Universal Robots PolyScope program: faichun_9jan_1t1.urp

Program faichun_9jan_1t1 (installation=default directory=/programs createdIn=5.11.9.1010452 lastSavedIn=5.11.9.1010452 robotSerialNumber=20225200364)
Calibrated DH parameters: a=[0.00002, -0.569483, -0.54992, -0.00001, -0.000036, 0]; d=[0.180894, -146.691669, 192.918669, -46.053088, 0.119778, 0.115602]; alpha=[1.571425, -0.001534, 0.003359, 1.568739, -1.571477, 0]; deltaTheta=[0, 0.376258, -0.101074, -0.275185, -0.000002, 0]
Robot Program (runOnlyOnce=true)
  Script file /programs/FaiChun_9 Jan_11_2_t1.script
    | def Machining1():
    |   # Default parameters:
    |   global speed_ms = 0.05
    |   global speed_rads = 0.75
    |   global accel_mss = 3
    |   global accel_radss = 1.2
    |   global blend_radius_m = 0.0003
    | 
    |   # Add subprograms here
    |   # Start of main program
    |   # Program generated by RoboDK v5.6.8 for UR10e on 17/01/2025 15:24:14
    |   # Using nominal kinematics.
    |   blend_radius_m = 0.0003
    |   speed_ms = 0.05
    |   # set_reference(p[0.340000, -0.240000, 0.001500, 0.000000, 0.000000, 0.000000])
    |   set_tcp(p[0.000000, 0.000000, 0.252000, 0.000000, 0.000000, 0.000000])
    |   # Show Tool
    |   movej([0.140721, -1.398447, -2.445688, -0.868253, 1.570796, 1.711517],accel_radss,speed_rads,0,blend_radius_m)
    |   movel([0.140721, -1.451124, -2.475554, -0.785711, 1.570796, 1.711517],accel_mss,speed_ms,0,blend_radius_m)
    |   #SetTool1
    |   #M_RunCode6
    |   #SetRPM60000
    |   speed_ms = 0.05
    |   #M_RunCode3
    |   movel([0.140721, -1.474076, -2.486639, -0.751674, 1.570796, 1.711517],accel_mss,speed_ms,0,blend_radius_m)
    |   speed_ms = 0.003
    |   movel([0.140721, -1.480003, -2.489338, -0.743048, 1.570796, 1.711517],accel_mss,speed_ms,0,blend_radius_m)
    |   speed_ms = 0.02
    |   movel([-0.135603, -1.563113, -2.412732, -0.736544, 1.570796, 1.435194],accel_mss,speed_ms,0,blend_radius_m)
    |   movel([-0.182919, -1.334068, -2.598334, -0.779987, 1.570796, 1.387878],accel_mss,speed_ms,0,blend_radius_m)
    |   movel([0.198662, -1.168946, -2.687374, -0.856069, 1.570796, 1.769459],accel_mss,speed_ms,0,blend_radius_m)
    |   movel([0.140721, -1.480003, -2.489338, -0.743048, 1.570796, 1.711517],accel_mss,speed_ms,0,blend_radius_m)
    |   speed_ms = 0.003
    |   movel([0.140721, -1.474076, -2.486639, -0.751674, 1.570796, 1.711517],accel_mss,speed_ms,0,blend_radius_m)
    |   speed_ms = 0.05
    |   movel([0.140721, -1.451124, -2.475554, -0.785711, 1.570796, 1.711517],accel_mss,speed_ms,0,blend_radius_m)
    |   #M_RunCode9
    |   movel([0.136570, -1.444454, -2.480985, -0.786951, 1.570796, 1.707367],accel_mss,speed_ms,0,blend_radius_m)
    |   #M_RunCode3
    |   movel([0.136570, -1.467543, -2.492148, -0.752698, 1.570796, 1.707367],accel_mss,speed_ms,0,blend_radius_m)
    |   speed_ms = 0.003
    |   movel([0.136570, -1.473508, -2.494867, -0.744014, 1.570796, 1.707367],accel_mss,speed_ms,0,blend_radius_m)
    |   speed_ms = 0.012
    |   movel([0.132210, -1.474416, -2.494098, -0.743875, 1.570796, 1.703007],accel_mss,speed_ms,0,blend_radius_m)
    |   movel([0.131633, -1.478168, -2.490906, -0.743314, 1.570796, 1.702429],accel_mss,speed_ms,0,blend_radius_m)
    |   movel([0.125209, -1.479526, -2.489746, -0.743117, 1.570796, 1.696006],accel_mss,speed_ms,0,blend_radius_m)
    |   movel([0.125756, -1.475786, -2.492935, -0.743668, 1.570796, 1.696552],accel_mss,speed_ms,0,blend_radius_m)
    |   movel([0.123495, -1.476273, -2.492521, -0.743595, 1.570796, 1.694292],accel_mss,speed_ms,0,blend_radius_m)
    |   movel([0.122957, -1.480010, -2.489332, -0.743047, 1.570796, 1.693753],accel_mss,speed_ms,0,blend_radius_m)
    |   movel([0.117581, -1.481181, -2.488328, -0.742880, 1.570796, 1.688377],accel_mss,speed_ms,0,blend_radius_m)
    |   movel([0.116539, -1.481408, -2.488133, -0.742848, 1.570796, 1.687335],accel_mss,speed_ms,0,blend_radius_m)
    |   movel([0.117294, -1.475890, -2.492847, -0.743652, 1.570796, 1.688091],accel_mss,speed_ms,0,blend_radius_m)
    |   movel([0.121657, -1.474929, -2.493663, -0.743797, 1.570796, 1.692454],accel_mss,speed_ms,0,blend_radius_m)
    |   movel([0.121935, -1.472979, -2.495315, -0.744096, 1.570796, 1.692731],accel_mss,speed_ms,0,blend_radius_m)
    |   movel([0.115294, -1.474450, -2.494069, -0.743870, 1.570796, 1.686091],accel_mss,speed_ms,0,blend_radius_m)
    |   movel([0.114291, -1.481907, -2.487705, -0.742777, 1.570796, 1.685087],accel_mss,speed_ms,0,blend_radius_m)
    |   movel([0.113249, -1.482141, -2.487504, -0.742744, 1.570796, 1.684045],accel_mss,speed_ms,0,blend_radius_m)
    |   speed_ms = 0.02
    |   movel([-0.001403, -1.512452, -2.460728, -0.739209, 1.570796, 1.569393],accel_mss,speed_ms,0,blend_radius_m)
    |   movel([-0.112335, -1.550651, -2.424918, -0.736820, 1.570796, 1.458461],accel_mss,speed_ms,0,blend_radius_m)
    |   speed_ms = 0.012
    |   movel([-0.113250, -1.544354, -2.430981, -0.737054, 1.570796, 1.457547],accel_mss,speed_ms,0,blend_radius_m)
    |   movel([-0.119333, -1.546716, -2.428713, -0.736959, 1.570796, 1.451463],accel_mss,speed_ms,0,blend_radius_m)
    |   movel([-0.119087, -1.548345, -2.427145, -0.736899, 1.570796, 1.451710],accel_mss,speed_ms,0,blend_radius_m)
    |   movel([-0.115090, -1.546793, -2.428639, -0.736956, 1.570796, 1.455706],accel_mss,speed_ms,0,blend_radius_m)
    |   movel([-0.114409, -1.551442, -2.424151, -0.736796, 1.570796, 1.456387],accel_mss,speed_ms,0,blend_radius_m)
    |   movel([-0.115366, -1.551811, -2.423794, -0.736784, 1.570796, 1.455430],accel_mss,speed_ms,0,blend_radius_m)
    |   movel([-0.120291, -1.553718, -2.421942, -0.736729, 1.570796, 1.450506],accel_mss,speed_ms,0,blend_radius_m)
    |   movel([-0.120772, -1.550599, -2.424968, -0.736822, 1.570796, 1.450025],accel_mss,speed_ms,0,blend_radius_m)
    |   movel([-0.122835, -1.551404, -2.424188, -0.736797, 1.570796, 1.447961],accel_mss,speed_ms,0,blend_radius_m)
    |   movel([-0.122346, -1.554519, -2.421162, -0.736708, 1.570796, 1.448450],accel_mss,speed_ms,0,blend_radius_m)
    |   movel([-0.128198, -1.556814, -2.418922, -0.736653, 1.570796, 1.442598],accel_mss,speed_ms,0,blend_radius_m)
    |   movel([-0.128709, -1.553718, -2.421941, -0.736729, 1.570796, 1.442088],accel_mss,speed_ms,0,blend_radius_m)
    |   movel([-0.132665, -1.555290, -2.420410, -0.736688, 1.570796, 1.438132],accel_mss,speed_ms,0,blend_radius_m)
    |   movel([-0.133450, -1.550705, -2.424865, -0.736819, 1.570796, 1.437347],accel_mss,speed_ms,0,blend_radius_m)
    |   movel([-0.129474, -1.549116, -2.426401, -0.736872, 1.570796, 1.441323],accel_mss,speed_ms,0,blend_radius_m)
    |   movel([-0.129743, -1.547498, -2.427961, -0.736930, 1.570796, 1.441053],accel_mss,speed_ms,0,blend_radius_m)
    |   movel([-0.133727, -1.549091, -2.426425, -0.736873, 1.570796, 1.437069],accel_mss,speed_ms,0,blend_radius_m)
    |   movel([-0.134396, -1.545231, -2.430140, -0.737018, 1.570796, 1.436400],accel_mss,speed_ms,0,blend_radius_m)
    |   movel([-0.134524, -1.544477, -2.430863, -0.737049, 1.570796, 1.436272],accel_mss,speed_ms,0,blend_radius_m)
    |   movel([-0.128589, -1.542092, -2.433143, -0.737154, 1.570796, 1.442208],accel_mss,speed_ms,0,blend_radius_m)
    |   movel([-0.128072, -1.545228, -2.430143, -0.737018, 1.570796, 1.442725],accel_mss,speed_ms,0,blend_radius_m)
    |   movel([-0.125992, -1.544401, -2.430936, -0.737052, 1.570796, 1.444805],accel_mss,speed_ms,0,blend_radius_m)
    |   movel([-0.126769, -1.539625, -2.435492, -0.737272, 1.570796, 1.444027],accel_mss,speed_ms,0,blend_radius_m)
    |   movel([-0.134806, -1.542853, -2.432416, -0.737120, 1.570796, 1.435990],accel_mss,speed_ms,0,blend_radius_m)
    |   movel([-0.151268, -1.454119, -2.510984, -0.747286, 1.570796, 1.419528],accel_mss,speed_ms,0,blend_radius_m)
    |   speed_ms = 0.02
    |   movel([-0.171874, -1.356528, -2.583560, -0.772301, 1.570796, 1.398922],accel_mss,speed_ms,0,blend_radius_m)
    |   movel([-0.172081, -1.355600, -2.584184, -0.772605, 1.570796, 1.398715],accel_mss,speed_ms,0,blend_radius_m)
    |   speed_ms = 0.012
    |   movel([-0.162028, -1.350393, -2.587664, -0.774332, 1.570796, 1.408769],accel_mss,speed_ms,0,blend_radius_m)
    |   movel([-0.163290, -1.344436, -2.591600, -0.776353, 1.570796, 1.407507],accel_mss,speed_ms,0,blend_radius_m)
    |   movel([-0.165922, -1.345805, -2.590700, -0.775884, 1.570796, 1.404874],accel_mss,speed_ms,0,blend_radius_m)
    |   movel([-0.165080, -1.349718, -2.588113, -0.774558, 1.570796, 1.405716],accel_mss,speed_ms,0,blend_radius_m)
    |   movel([-0.172527, -1.353588, -2.585533, -0.773268, 1.570796, 1.398269],accel_mss,speed_ms,0,blend_radius_m)
    |   movel([-0.172737, -1.352660, -2.586154, -0.773575, 1.570796, 1.398059],accel_mss,speed_ms,0,blend_radius_m)
    |   movel([-0.173831, -1.347848, -2.589351, -0.775189, 1.570796, 1.396966],accel_mss,speed_ms,0,blend_radius_m)
    |   movel([-0.168773, -1.345194, -2.591101, -0.776093, 1.570796, 1.402023],accel_mss,speed_ms,0,blend_radius_m)
    |   movel([-0.169223, -1.343160, -2.592436, -0.776792, 1.570796, 1.401574],accel_mss,speed_ms,0,blend_radius_m)
    |   movel([-0.174292, -1.345828, -2.590684, -0.775876, 1.570796, 1.396505],accel_mss,speed_ms,0,blend_radius_m)
    |   movel([-0.175621, -1.340037, -2.594475, -0.777877, 1.570796, 1.395175],accel_mss,speed_ms,0,blend_radius_m)
    |   movel([-0.170518, -1.337328, -2.596232, -0.778829, 1.570796, 1.400279],accel_mss,speed_ms,0,blend_radius_m)
    |   movel([-0.171402, -1.333368, -2.598783, -0.780238, 1.570796, 1.399394],accel_mss,speed_ms,0,blend_radius_m)
    |   movel([-0.163769, -1.329319, -2.601369, -0.781700, 1.570796, 1.407028],accel_mss,speed_ms,0,blend_radius_m)
    |   movel([-0.162919, -1.333321, -2.598813, -0.780255, 1.570796, 1.407878],accel_mss,speed_ms,0,blend_radius_m)
    |   movel([-0.160246, -1.331919, -2.599711, -0.780759, 1.570796, 1.410551],accel_mss,speed_ms,0,blend_radius_m)
    |   movel([-0.161083, -1.327903, -2.602269, -0.782217, 1.570796, 1.409713],accel_mss,speed_ms,0,blend_radius_m)
    |   movel([-0.153386, -1.323865, -2.604819, -0.783706, 1.570796, 1.417410],accel_mss,speed_ms,0,blend_radius_m)
    |   movel([-0.152202, -1.329868, -2.601020, -0.781501, 1.570796, 1.418594],accel_mss,speed_ms,0,blend_radius_m)
    |   movel([-0.157369, -1.332552, -2.599306, -0.780531, 1.570796, 1.413427],accel_mss,speed_ms,0,blend_radius_m)
    |   movel([-0.156945, -1.334634, -2.597970, -0.779785, 1.570796, 1.413851],accel_mss,speed_ms,0,blend_radius_m)
    |   movel([-0.149106, -1.330580, -2.600566, -0.781243, 1.570796, 1.421690],accel_mss,speed_ms,0,blend_radius_m)
    |   movel([-0.150679, -1.322452, -2.605705, -0.784232, 1.570796, 1.420118],accel_mss,speed_ms,0,blend_radius_m)
    |   movel([-0.001924, -1.251119, -2.647144, -0.814126, 1.570796, 1.568873],accel_mss,speed_ms,0,blend_radius_m)
    |   speed_ms = 0.02
    |   movel([0.158957, -1.188696, -2.678386, -0.845308, 1.570796, 1.729754],accel_mss,speed_ms,0,blend_radius_m)
    |   movel([0.157034, -1.200160, -2.672976, -0.839253, 1.570796, 1.727831],accel_mss,speed_ms,0,blend_radius_m)
    |   speed_ms = 0.012
    |   movel([0.166189, -1.197160, -2.674405, -0.840823, 1.570796, 1.736986],accel_mss,speed_ms,0,blend_radius_m)
    |   movel([0.166716, -1.194184, -2.675814, -0.842391, 1.570796, 1.737513],accel_mss,speed_ms,0,blend_radius_m)
    |   movel([0.160669, -1.196167, -2.674876, -0.841345, 1.570796, 1.731466],accel_mss,speed_ms,0,blend_radius_m)
    |   movel([0.162134, -1.187639, -2.678877, -0.845873, 1.570796, 1.732930],accel_mss,speed_ms,0,blend_radius_m)
    |   movel([0.163603, -1.187149, -2.679104, -0.846136, 1.570796, 1.734399],accel_mss,speed_ms,0,blend_radius_m)
    |   movel([0.171178, -1.184645, -2.680263, -0.847481, 1.570796, 1.741974],accel_mss,speed_ms,0,blend_radius_m)
    |   movel([0.170131, -1.190457, -2.677564, -0.844368, 1.570796, 1.740927],accel_mss,speed_ms,0,blend_radius_m)
    |   movel([0.173284, -1.189438, -2.678039, -0.844911, 1.570796, 1.744080],accel_mss,speed_ms,0,blend_radius_m)
    |   movel([0.174358, -1.183606, -2.680741, -0.848041, 1.570796, 1.745154],accel_mss,speed_ms,0,blend_radius_m)
    |   movel([0.183424, -1.180682, -2.682083, -0.849624, 1.570796, 1.754220],accel_mss,speed_ms,0,blend_radius_m)
    |   movel([0.182294, -1.186557, -2.679379, -0.846453, 1.570796, 1.753091],accel_mss,speed_ms,0,blend_radius_m)
    |   movel([0.188385, -1.184641, -2.680265, -0.847483, 1.570796, 1.759181],accel_mss,speed_ms,0,blend_radius_m)
    |   movel([0.186680, -1.193280, -2.676240, -0.842870, 1.570796, 1.757477],accel_mss,speed_ms,0,blend_radius_m)
    |   movel([0.180648, -1.195154, -2.675356, -0.841879, 1.570796, 1.751444],accel_mss,speed_ms,0,blend_radius_m)
    |   movel([0.180078, -1.198139, -2.673940, -0.840310, 1.570796, 1.750875],accel_mss,speed_ms,0,blend_radius_m)
    |   movel([0.186090, -1.196283, -2.674822, -0.841285, 1.570796, 1.756886],accel_mss,speed_ms,0,blend_radius_m)
    |   movel([0.184696, -1.203394, -2.671424, -0.837571, 1.570796, 1.755493],accel_mss,speed_ms,0,blend_radius_m)
    |   movel([0.184428, -1.204765, -2.670763, -0.836861, 1.570796, 1.755225],accel_mss,speed_ms,0,blend_radius_m)
    |   movel([0.175610, -1.207468, -2.669453, -0.835468, 1.570796, 1.746407],accel_mss,speed_ms,0,blend_radius_m)
    |   movel([0.176673, -1.201793, -2.672194, -0.838402, 1.570796, 1.747469],accel_mss,speed_ms,0,blend_radius_m)
    |   movel([0.173563, -1.202767, -2.671726, -0.837896, 1.570796, 1.744359],accel_mss,speed_ms,0,blend_radius_m)
    |   movel([0.171983, -1.211350, -2.667557, -0.833482, 1.570796, 1.742780],accel_mss,speed_ms,0,blend_radius_m)
    |   movel([0.183853, -1.207714, -2.669333, -0.835342, 1.570796, 1.754649],accel_mss,speed_ms,0,blend_radius_m)
    |   speed_ms = 0.02
    |   movel([0.158243, -1.345021, -2.591215, -0.776152, 1.570796, 1.729039],accel_mss,speed_ms,0,blend_radius_m)
    |   movel([0.139022, -1.458254, -2.507595, -0.746540, 1.570796, 1.709818],accel_mss,speed_ms,0,blend_radius_m)
    |   speed_ms = 0.012
    |   movel([0.130132, -1.460164, -2.506021, -0.746204, 1.570796, 1.700928],accel_mss,speed_ms,0,blend_radius_m)
    |   movel([0.129256, -1.465966, -2.501205, -0.745218, 1.570796, 1.700052],accel_mss,speed_ms,0,blend_radius_m)
    |   movel([0.131545, -1.465473, -2.501616, -0.745300, 1.570796, 1.702341],accel_mss,speed_ms,0,blend_radius_m)
    |   movel([0.132131, -1.461656, -2.504788, -0.745945, 1.570796, 1.702927],accel_mss,speed_ms,0,blend_radius_m)
    |   movel([0.138690, -1.460258, -2.505944, -0.746187, 1.570796, 1.709487],accel_mss,speed_ms,0,blend_radius_m)
    |   movel([0.138542, -1.461182, -2.505180, -0.746027, 1.570796, 1.709338],accel_mss,speed_ms,0,blend_radius_m)
    |   movel([0.137780, -1.465926, -2.501239, -0.745225, 1.570796, 1.708576],accel_mss,speed_ms,0,blend_radius_m)
    |   movel([0.133380, -1.466851, -2.500465, -0.745072, 1.570796, 1.704177],accel_mss,speed_ms,0,blend_radius_m)
    |   movel([0.133075, -1.468822, -2.498815, -0.744752, 1.570796, 1.703871],accel_mss,speed_ms,0,blend_radius_m)
    |   movel([0.137466, -1.467900, -2.499588, -0.744901, 1.570796, 1.708263],accel_mss,speed_ms,0,blend_radius_m)
    |   movel([0.136570, -1.473508, -2.494867, -0.744014, 1.570796, 1.707367],accel_mss,speed_ms,0,blend_radius_m)
    |   speed_ms = 0.003
    |   movel([0.136570, -1.467543, -2.492148, -0.752698, 1.570796, 1.707367],accel_mss,speed_ms,0,blend_radius_m)
    |   speed_ms = 0.05
    |   movel([0.136570, -1.444454, -2.480985, -0.786951, 1.570796, 1.707367],accel_mss,speed_ms,0,blend_radius_m)
    |   #M_RunCode9
    |   movel([-0.101116, -1.322556, -2.569102, -0.820731, 1.570796, 1.469680],accel_mss,speed_ms,0,blend_radius_m)
    |   #M_RunCode3
    |   # num 0 inside
    |   movel([-0.101116, -1.347956, -2.581781, -0.782652, 1.570796, 1.469680],accel_mss,speed_ms,0,blend_radius_m)
    |   speed_ms = 0.003
    |   movel([-0.101116, -1.354564, -2.584879, -0.772945, 1.570796, 1.469680],accel_mss,speed_ms,0,blend_radius_m)
    |   speed_ms = 0.015
    |   movel([-0.106161, -1.361335, -2.580307, -0.770747, 1.570796, 1.464635],accel_mss,speed_ms,0,blend_radius_m)
    |   movel([-0.110090, -1.365943, -2.577159, -0.769287, 1.570796, 1.460707],accel_mss,speed_ms,0,blend_radius_m)
    |   movel([-0.111700, -1.367455, -2.576119, -0.768814, 1.570796, 1.459096],accel_mss,speed_ms,0,blend_radius_m)
    |   movel([-0.113150, -1.368443, -2.575438, -0.768507, 1.570796, 1.457647],accel_mss,speed_ms,0,blend_radius_m)
    |   movel([-0.114438, -1.368913, -2.575114, -0.768362, 1.570796, 1.456358],accel_mss,speed_ms,0,blend_radius_m)
    |   movel([-0.115571, -1.368864, -2.575148, -0.768377, 1.570796, 1.455226],accel_mss,speed_ms,0,blend_radius_m)
    |   movel([-0.116374, -1.368348, -2.575504, -0.768537, 1.570796, 1.454422],accel_mss,speed_ms,0,blend_radius_m)
    |   movel([-0.116674, -1.367414, -2.576148, -0.768827, 1.570796, 1.454122],accel_mss,speed_ms,0,blend_radius_m)
    |   movel([-0.116470, -1.366059, -2.577080, -0.769251, 1.570796, 1.454326],accel_mss,speed_ms,0,blend_radius_m)
    |   movel([-0.115761, -1.364279, -2.578299, -0.769810, 1.570796, 1.455035],accel_mss,speed_ms,0,blend_radius_m)
    |   movel([-0.112933, -1.359327, -2.581670, -0.771392, 1.570796, 1.457863],accel_mss,speed_ms,0,blend_radius_m)
    |   movel([-0.108281, -1.352413, -2.586319, -0.773657, 1.570796, 1.462515],accel_mss,speed_ms,0,blend_radius_m)
    |   movel([-0.103194, -1.345531, -2.590880, -0.775978, 1.570796, 1.467603],accel_mss,speed_ms,0,blend_radius_m)
    |   movel([-0.099141, -1.340763, -2.594002, -0.777624, 1.570796, 1.471655],accel_mss,speed_ms,0,blend_radius_m)
    |   movel([-0.097464, -1.339187, -2.595027, -0.778175, 1.570796, 1.473333],accel_mss,speed_ms,0,blend_radius_m)
    |   movel([-0.095957, -1.338153, -2.595698, -0.778538, 1.570796, 1.474840],accel_mss,speed_ms,0,blend_radius_m)
    |   movel([-0.094620, -1.337665, -2.596014, -0.778710, 1.570796, 1.476176],accel_mss,speed_ms,0,blend_radius_m)
    |   movel([-0.093457, -1.337724, -2.595976, -0.778689, 1.570796, 1.477339],accel_mss,speed_ms,0,blend_radius_m)
    |   movel([-0.092647, -1.338276, -2.595618, -0.778495, 1.570796, 1.478149],accel_mss,speed_ms,0,blend_radius_m)
    |   movel([-0.092365, -1.339263, -2.594978, -0.778148, 1.570796, 1.478432],accel_mss,speed_ms,0,blend_radius_m)
    |   movel([-0.092614, -1.340685, -2.594053, -0.777651, 1.570796, 1.478183],accel_mss,speed_ms,0,blend_radius_m)
    |   movel([-0.093386, -1.342532, -2.592847, -0.777009, 1.570796, 1.477410],accel_mss,speed_ms,0,blend_radius_m)
    |   movel([-0.096363, -1.347612, -2.589507, -0.775269, 1.570796, 1.474433],accel_mss,speed_ms,0,blend_radius_m)
    |   movel([-0.101116, -1.354564, -2.584879, -0.772945, 1.570796, 1.469680],accel_mss,speed_ms,0,blend_radius_m)
    |   speed_ms = 0.003
    |   movel([-0.101116, -1.347956, -2.581781, -0.782652, 1.570796, 1.469680],accel_mss,speed_ms,0,blend_radius_m)
    |   speed_ms = 0.05
    |   movel([-0.101116, -1.322556, -2.569102, -0.820731, 1.570796, 1.469680],accel_mss,speed_ms,0,blend_radius_m)
    |   #M_RunCode9
    |   movel([-0.093439, -1.325002, -2.567533, -0.819854, 1.570796, 1.477357],accel_mss,speed_ms,0,blend_radius_m)
    |   #M_RunCode3
    |   #num 0 outside
    |   movel([-0.093439, -1.350361, -2.580180, -0.781848, 1.570796, 1.477357],accel_mss,speed_ms,0,blend_radius_m)
    |   speed_ms = 0.003
    |   movel([-0.093439, -1.356958, -2.583270, -0.772161, 1.570796, 1.477357],accel_mss,speed_ms,0,blend_radius_m)
    |   speed_ms = 0.015
    |   movel([-0.095323, -1.359406, -2.581617, -0.771367, 1.570796, 1.475474],accel_mss,speed_ms,0,blend_radius_m)
    |   movel([-0.097250, -1.361605, -2.580124, -0.770660, 1.570796, 1.473546],accel_mss,speed_ms,0,blend_radius_m)
    |   movel([-0.099225, -1.363562, -2.578790, -0.770037, 1.570796, 1.471571],accel_mss,speed_ms,0,blend_radius_m)
    |   movel([-0.101247, -1.365276, -2.577617, -0.769496, 1.570796, 1.469549],accel_mss,speed_ms,0,blend_radius_m)
    |   movel([-0.103277, -1.366737, -2.576613, -0.769038, 1.570796, 1.467519],accel_mss,speed_ms,0,blend_radius_m)
    |   movel([-0.105274, -1.367936, -2.575788, -0.768665, 1.570796, 1.465522],accel_mss,speed_ms,0,blend_radius_m)
    |   movel([-0.107241, -1.368876, -2.575140, -0.768373, 1.570796, 1.463555],accel_mss,speed_ms,0,blend_radius_m)
    |   movel([-0.109177, -1.369553, -2.574672, -0.768164, 1.570796, 1.461619],accel_mss,speed_ms,0,blend_radius_m)
    |   movel([-0.111057, -1.369973, -2.574381, -0.768035, 1.570796, 1.459739],accel_mss,speed_ms,0,blend_radius_m)
    |   movel([-0.112847, -1.370143, -2.574264, -0.767982, 1.570796, 1.457949],accel_mss,speed_ms,0,blend_radius_m)
    |   movel([-0.114554, -1.370059, -2.574322, -0.768008, 1.570796, 1.456243],accel_mss,speed_ms,0,blend_radius_m)
    |   movel([-0.116176, -1.369726, -2.574552, -0.768111, 1.570796, 1.454621],accel_mss,speed_ms,0,blend_radius_m)
    |   movel([-0.117639, -1.369161, -2.574943, -0.768285, 1.570796, 1.453158],accel_mss,speed_ms,0,blend_radius_m)
    |   movel([-0.118861, -1.368389, -2.575476, -0.768524, 1.570796, 1.451935],accel_mss,speed_ms,0,blend_radius_m)
    |   movel([-0.119847, -1.367410, -2.576151, -0.768828, 1.570796, 1.450949],accel_mss,speed_ms,0,blend_radius_m)
    |   movel([-0.120593, -1.366216, -2.576972, -0.769201, 1.570796, 1.450203],accel_mss,speed_ms,0,blend_radius_m)
    |   movel([-0.121076, -1.364824, -2.577927, -0.769639, 1.570796, 1.449720],accel_mss,speed_ms,0,blend_radius_m)
    |   movel([-0.121271, -1.363244, -2.579007, -0.770138, 1.570796, 1.449525],accel_mss,speed_ms,0,blend_radius_m)
    |   movel([-0.121177, -1.361471, -2.580215, -0.770703, 1.570796, 1.449619],accel_mss,speed_ms,0,blend_radius_m)
    |   movel([-0.120789, -1.359505, -2.581549, -0.771335, 1.570796, 1.450007],accel_mss,speed_ms,0,blend_radius_m)
    |   movel([-0.120098, -1.357373, -2.582991, -0.772026, 1.570796, 1.450698],accel_mss,speed_ms,0,blend_radius_m)
    |   movel([-0.119085, -1.355103, -2.584518, -0.772768, 1.570796, 1.451711],accel_mss,speed_ms,0,blend_radius_m)
    |   movel([-0.117751, -1.352697, -2.586129, -0.773563, 1.570796, 1.453045],accel_mss,speed_ms,0,blend_radius_m)
    |   movel([-0.116093, -1.350152, -2.587824, -0.774413, 1.570796, 1.454704],accel_mss,speed_ms,0,blend_radius_m)
    |   movel([-0.114233, -1.347648, -2.589484, -0.775257, 1.570796, 1.456564],accel_mss,speed_ms,0,blend_radius_m)
    |   movel([-0.112304, -1.345376, -2.590982, -0.776031, 1.570796, 1.458493],accel_mss,speed_ms,0,blend_radius_m)
    |   movel([-0.110305, -1.343337, -2.592320, -0.776731, 1.570796, 1.460492],accel_mss,speed_ms,0,blend_radius_m)
    |   movel([-0.108239, -1.341537, -2.593498, -0.777355, 1.570796, 1.462557],accel_mss,speed_ms,0,blend_radius_m)
    |   movel([-0.106152, -1.339991, -2.594504, -0.777893, 1.570796, 1.464644],accel_mss,speed_ms,0,blend_radius_m)
    |   movel([-0.104092, -1.338723, -2.595328, -0.778337, 1.570796, 1.466704],accel_mss,speed_ms,0,blend_radius_m)
    |   movel([-0.102059, -1.337730, -2.595972, -0.778687, 1.570796, 1.468737],accel_mss,speed_ms,0,blend_radius_m)
    |   movel([-0.100055, -1.337017, -2.596433, -0.778939, 1.570796, 1.470741],accel_mss,speed_ms,0,blend_radius_m)
    |   movel([-0.098115, -1.336579, -2.596716, -0.779094, 1.570796, 1.472681],accel_mss,speed_ms,0,blend_radius_m)
    |   movel([-0.096266, -1.336409, -2.596826, -0.779154, 1.570796, 1.474530],accel_mss,speed_ms,0,blend_radius_m)
    |   movel([-0.094508, -1.336506, -2.596763, -0.779120, 1.570796, 1.476288],accel_mss,speed_ms,0,blend_radius_m)
    |   movel([-0.092848, -1.336874, -2.596526, -0.778989, 1.570796, 1.477948],accel_mss,speed_ms,0,blend_radius_m)
    |   movel([-0.091363, -1.337486, -2.596130, -0.778773, 1.570796, 1.479434],accel_mss,speed_ms,0,blend_radius_m)
    |   movel([-0.090132, -1.338313, -2.595594, -0.778482, 1.570796, 1.480664],accel_mss,speed_ms,0,blend_radius_m)
    |   movel([-0.089156, -1.339357, -2.594917, -0.778115, 1.570796, 1.481641],accel_mss,speed_ms,0,blend_radius_m)
    |   movel([-0.088434, -1.340616, -2.594098, -0.777675, 1.570796, 1.482363],accel_mss,speed_ms,0,blend_radius_m)
    |   movel([-0.087990, -1.342075, -2.593146, -0.777168, 1.570796, 1.482806],accel_mss,speed_ms,0,blend_radius_m)
    |   movel([-0.087851, -1.343724, -2.592067, -0.776598, 1.570796, 1.482946],accel_mss,speed_ms,0,blend_radius_m)
    |   movel([-0.088015, -1.345563, -2.590859, -0.775967, 1.570796, 1.482781],accel_mss,speed_ms,0,blend_radius_m)
    |   movel([-0.088479, -1.347585, -2.589526, -0.775279, 1.570796, 1.482317],accel_mss,speed_ms,0,blend_radius_m)
    |   movel([-0.089250, -1.349756, -2.588088, -0.774546, 1.570796, 1.481546],accel_mss,speed_ms,0,blend_radius_m)
    |   movel([-0.090337, -1.352044, -2.586565, -0.773780, 1.570796, 1.480459],accel_mss,speed_ms,0,blend_radius_m)
    |   movel([-0.091734, -1.354445, -2.584959, -0.772985, 1.570796, 1.479062],accel_mss,speed_ms,0,blend_radius_m)
    |   movel([-0.093439, -1.356958, -2.583270, -0.772161, 1.570796, 1.477357],accel_mss,speed_ms,0,blend_radius_m)
    |   speed_ms = 0.003
    |   movel([-0.093439, -1.350361, -2.580180, -0.781848, 1.570796, 1.477357],accel_mss,speed_ms,0,blend_radius_m)
    |   speed_ms = 0.05
    |   movel([-0.093439, -1.325002, -2.567533, -0.819854, 1.570796, 1.477357],accel_mss,speed_ms,0,blend_radius_m)
    |   #M_RunCode9
    |   movel([-0.123954, -1.324456, -2.567884, -0.820049, 1.570796, 1.446843],accel_mss,speed_ms,0,blend_radius_m)
    |   #M_RunCode3
    |   # num 2
    |   movel([-0.123954, -1.349824, -2.580538, -0.782027, 1.570796, 1.446843],accel_mss,speed_ms,0,blend_radius_m)
    |   speed_ms = 0.003
    |   movel([-0.123954, -1.356423, -2.583630, -0.772335, 1.570796, 1.446843],accel_mss,speed_ms,0,blend_radius_m)
    |   speed_ms = 0.02
    |   movel([-0.129998, -1.365194, -2.577673, -0.769522, 1.570796, 1.440798],accel_mss,speed_ms,0,blend_radius_m)
    |   movel([-0.153716, -1.359168, -2.581778, -0.771443, 1.570796, 1.417080],accel_mss,speed_ms,0,blend_radius_m)
    |   movel([-0.153133, -1.358284, -2.582375, -0.771729, 1.570796, 1.417664],accel_mss,speed_ms,0,blend_radius_m)
    |   movel([-0.151367, -1.356095, -2.583852, -0.772443, 1.570796, 1.419429],accel_mss,speed_ms,0,blend_radius_m)
    |   movel([-0.149072, -1.354075, -2.585207, -0.773107, 1.570796, 1.421725],accel_mss,speed_ms,0,blend_radius_m)
    |   movel([-0.146447, -1.352249, -2.586428, -0.773712, 1.570796, 1.424349],accel_mss,speed_ms,0,blend_radius_m)
    |   movel([-0.143702, -1.350644, -2.587497, -0.774248, 1.570796, 1.427094],accel_mss,speed_ms,0,blend_radius_m)
    |   movel([-0.136140, -1.346869, -2.589998, -0.775522, 1.570796, 1.434656],accel_mss,speed_ms,0,blend_radius_m)
    |   movel([-0.129079, -1.343432, -2.592258, -0.776699, 1.570796, 1.441717],accel_mss,speed_ms,0,blend_radius_m)
    |   movel([-0.126471, -1.341951, -2.593227, -0.777211, 1.570796, 1.444325],accel_mss,speed_ms,0,blend_radius_m)
    |   movel([-0.124017, -1.340294, -2.594308, -0.777788, 1.570796, 1.446780],accel_mss,speed_ms,0,blend_radius_m)
    |   movel([-0.121890, -1.338487, -2.595482, -0.778421, 1.570796, 1.448906],accel_mss,speed_ms,0,blend_radius_m)
    |   movel([-0.120264, -1.336553, -2.596733, -0.779103, 1.570796, 1.450532],accel_mss,speed_ms,0,blend_radius_m)
    |   movel([-0.118963, -1.334098, -2.598315, -0.779977, 1.570796, 1.451833],accel_mss,speed_ms,0,blend_radius_m)
    |   movel([-0.118722, -1.333042, -2.598992, -0.780355, 1.570796, 1.452075],accel_mss,speed_ms,0,blend_radius_m)
    |   movel([-0.118753, -1.332102, -2.599594, -0.780693, 1.570796, 1.452044],accel_mss,speed_ms,0,blend_radius_m)
    |   movel([-0.119446, -1.330656, -2.600518, -0.781215, 1.570796, 1.451350],accel_mss,speed_ms,0,blend_radius_m)
    |   movel([-0.120855, -1.329858, -2.601026, -0.781505, 1.570796, 1.449941],accel_mss,speed_ms,0,blend_radius_m)
    |   movel([-0.122064, -1.329696, -2.601129, -0.781563, 1.570796, 1.448732],accel_mss,speed_ms,0,blend_radius_m)
    |   movel([-0.123171, -1.329886, -2.601009, -0.781495, 1.570796, 1.447625],accel_mss,speed_ms,0,blend_radius_m)
    |   movel([-0.124102, -1.330365, -2.600703, -0.781321, 1.570796, 1.446695],accel_mss,speed_ms,0,blend_radius_m)
    |   movel([-0.124778, -1.331064, -2.600258, -0.781068, 1.570796, 1.446018],accel_mss,speed_ms,0,blend_radius_m)
    |   movel([-0.125119, -1.332265, -2.599490, -0.780634, 1.570796, 1.445678],accel_mss,speed_ms,0,blend_radius_m)
    |   movel([-0.125345, -1.333426, -2.598746, -0.780217, 1.570796, 1.445451],accel_mss,speed_ms,0,blend_radius_m)
    |   movel([-0.126105, -1.334850, -2.597831, -0.779708, 1.570796, 1.444691],accel_mss,speed_ms,0,blend_radius_m)
    |   movel([-0.127495, -1.336400, -2.596832, -0.779157, 1.570796, 1.443301],accel_mss,speed_ms,0,blend_radius_m)
    |   movel([-0.129163, -1.337385, -2.596195, -0.778809, 1.570796, 1.441634],accel_mss,speed_ms,0,blend_radius_m)
    |   movel([-0.130909, -1.337812, -2.595919, -0.778658, 1.570796, 1.439887],accel_mss,speed_ms,0,blend_radius_m)
    |   movel([-0.132535, -1.337687, -2.596000, -0.778702, 1.570796, 1.438262],accel_mss,speed_ms,0,blend_radius_m)
    |   movel([-0.133822, -1.337065, -2.596402, -0.778922, 1.570796, 1.436975],accel_mss,speed_ms,0,blend_radius_m)
    |   movel([-0.134561, -1.335997, -2.597092, -0.779300, 1.570796, 1.436235],accel_mss,speed_ms,0,blend_radius_m)
    |   movel([-0.134602, -1.334568, -2.598012, -0.779809, 1.570796, 1.436194],accel_mss,speed_ms,0,blend_radius_m)
    |   movel([-0.133790, -1.332863, -2.599107, -0.780419, 1.570796, 1.437007],accel_mss,speed_ms,0,blend_radius_m)
    |   movel([-0.132656, -1.331465, -2.600001, -0.780923, 1.570796, 1.438141],accel_mss,speed_ms,0,blend_radius_m)
    |   movel([-0.131309, -1.330326, -2.600728, -0.781335, 1.570796, 1.439487],accel_mss,speed_ms,0,blend_radius_m)
    |   movel([-0.129748, -1.329445, -2.601289, -0.781655, 1.570796, 1.441048],accel_mss,speed_ms,0,blend_radius_m)
    |   movel([-0.127974, -1.328829, -2.601681, -0.781879, 1.570796, 1.442823],accel_mss,speed_ms,0,blend_radius_m)
    |   movel([-0.126079, -1.328474, -2.601907, -0.782009, 1.570796, 1.444717],accel_mss,speed_ms,0,blend_radius_m)
    |   movel([-0.124154, -1.328370, -2.601972, -0.782047, 1.570796, 1.446642],accel_mss,speed_ms,0,blend_radius_m)
    |   movel([-0.120221, -1.328934, -2.601614, -0.781841, 1.570796, 1.450575],accel_mss,speed_ms,0,blend_radius_m)
    |   movel([-0.117965, -1.329713, -2.601118, -0.781557, 1.570796, 1.452832],accel_mss,speed_ms,0,blend_radius_m)
    |   movel([-0.116035, -1.330744, -2.600461, -0.781183, 1.570796, 1.454762],accel_mss,speed_ms,0,blend_radius_m)
    |   movel([-0.114434, -1.332023, -2.599645, -0.780721, 1.570796, 1.456362],accel_mss,speed_ms,0,blend_radius_m)
    |   movel([-0.113162, -1.333549, -2.598667, -0.780173, 1.570796, 1.457634],accel_mss,speed_ms,0,blend_radius_m)
    |   movel([-0.112422, -1.335319, -2.597529, -0.779541, 1.570796, 1.458375],accel_mss,speed_ms,0,blend_radius_m)
    |   movel([-0.112423, -1.337340, -2.596224, -0.778825, 1.570796, 1.458373],accel_mss,speed_ms,0,blend_radius_m)
    |   movel([-0.113159, -1.339605, -2.594755, -0.778028, 1.570796, 1.457637],accel_mss,speed_ms,0,blend_radius_m)
    |   movel([-0.114621, -1.342110, -2.593123, -0.777156, 1.570796, 1.456175],accel_mss,speed_ms,0,blend_radius_m)
    |   movel([-0.116384, -1.344285, -2.591699, -0.776405, 1.570796, 1.454412],accel_mss,speed_ms,0,blend_radius_m)
    |   movel([-0.118449, -1.346179, -2.590453, -0.775757, 1.570796, 1.452347],accel_mss,speed_ms,0,blend_radius_m)
    |   movel([-0.120701, -1.347816, -2.589373, -0.775200, 1.570796, 1.450095],accel_mss,speed_ms,0,blend_radius_m)
    |   movel([-0.123019, -1.349217, -2.588445, -0.774727, 1.570796, 1.447777],accel_mss,speed_ms,0,blend_radius_m)
    |   movel([-0.128882, -1.352127, -2.586509, -0.773752, 1.570796, 1.441914],accel_mss,speed_ms,0,blend_radius_m)
    |   movel([-0.134390, -1.354902, -2.584653, -0.772834, 1.570796, 1.436406],accel_mss,speed_ms,0,blend_radius_m)
    |   movel([-0.136479, -1.356170, -2.583801, -0.772418, 1.570796, 1.434317],accel_mss,speed_ms,0,blend_radius_m)
    |   movel([-0.138470, -1.357620, -2.582824, -0.771945, 1.570796, 1.432326],accel_mss,speed_ms,0,blend_radius_m)
    |   movel([-0.140252, -1.359262, -2.581714, -0.771413, 1.570796, 1.430544],accel_mss,speed_ms,0,blend_radius_m)
    |   movel([-0.141709, -1.361091, -2.580474, -0.770825, 1.570796, 1.429087],accel_mss,speed_ms,0,blend_radius_m)
    |   movel([-0.140820, -1.361317, -2.580320, -0.770752, 1.570796, 1.429976],accel_mss,speed_ms,0,blend_radius_m)
    |   movel([-0.138271, -1.361815, -2.579981, -0.770593, 1.570796, 1.432526],accel_mss,speed_ms,0,blend_radius_m)
    |   movel([-0.135841, -1.361968, -2.579877, -0.770544, 1.570796, 1.434956],accel_mss,speed_ms,0,blend_radius_m)
    |   movel([-0.133532, -1.361779, -2.580005, -0.770605, 1.570796, 1.437265],accel_mss,speed_ms,0,blend_radius_m)
    |   movel([-0.131335, -1.361242, -2.580371, -0.770776, 1.570796, 1.439461],accel_mss,speed_ms,0,blend_radius_m)
    |   movel([-0.129273, -1.360410, -2.580936, -0.771043, 1.570796, 1.441523],accel_mss,speed_ms,0,blend_radius_m)
    |   movel([-0.127356, -1.359331, -2.581667, -0.771391, 1.570796, 1.443441],accel_mss,speed_ms,0,blend_radius_m)
    |   movel([-0.125585, -1.358004, -2.582565, -0.771820, 1.570796, 1.445212],accel_mss,speed_ms,0,blend_radius_m)
    |   movel([-0.123954, -1.356423, -2.583630, -0.772335, 1.570796, 1.446843],accel_mss,speed_ms,0,blend_radius_m)
    |   speed_ms = 0.003
    |   movel([-0.123954, -1.349824, -2.580538, -0.782027, 1.570796, 1.446843],accel_mss,speed_ms,0,blend_radius_m)
    |   speed_ms = 0.05
    |   movel([-0.123954, -1.324456, -2.567884, -0.820049, 1.570796, 1.446843],accel_mss,speed_ms,0,blend_radius_m)
    |   #M_RunCode9
    |   movel([0.068760, -1.419496, -2.500728, -0.792166, 1.570796, 1.639556],accel_mss,speed_ms,0,blend_radius_m)
    |   #M_RunCode3
    |   movel([0.068760, -1.443093, -2.512190, -0.757106, 1.570796, 1.639556],accel_mss,speed_ms,0,blend_radius_m)
    |   speed_ms = 0.003
    |   movel([0.068760, -1.449197, -2.514984, -0.748208, 1.570796, 1.639556],accel_mss,speed_ms,0,blend_radius_m)
    |   speed_ms = 0.02
    |   movel([0.070663, -1.447541, -2.516321, -0.748527, 1.570796, 1.641460],accel_mss,speed_ms,0,blend_radius_m)
    |   movel([0.072941, -1.446164, -2.517430, -0.748795, 1.570796, 1.643737],accel_mss,speed_ms,0,blend_radius_m)
    |   movel([0.075428, -1.445044, -2.518330, -0.749016, 1.570796, 1.646225],accel_mss,speed_ms,0,blend_radius_m)
    |   movel([0.077955, -1.444162, -2.519036, -0.749190, 1.570796, 1.648751],accel_mss,speed_ms,0,blend_radius_m)
    |   movel([0.084751, -1.442342, -2.520492, -0.749555, 1.570796, 1.655547],accel_mss,speed_ms,0,blend_radius_m)
    |   movel([0.091060, -1.440730, -2.521777, -0.749882, 1.570796, 1.661856],accel_mss,speed_ms,0,blend_radius_m)
    |   movel([0.093434, -1.439943, -2.522403, -0.750043, 1.570796, 1.664230],accel_mss,speed_ms,0,blend_radius_m)
    |   movel([0.095728, -1.438957, -2.523186, -0.750246, 1.570796, 1.666524],accel_mss,speed_ms,0,blend_radius_m)
    |   movel([0.097799, -1.437760, -2.524135, -0.750494, 1.570796, 1.668595],accel_mss,speed_ms,0,blend_radius_m)
    |   movel([0.099508, -1.436334, -2.525261, -0.750793, 1.570796, 1.670304],accel_mss,speed_ms,0,blend_radius_m)
    |   movel([0.101083, -1.434354, -2.526822, -0.751213, 1.570796, 1.671879],accel_mss,speed_ms,0,blend_radius_m)
    |   movel([0.101514, -1.433430, -2.527547, -0.751411, 1.570796, 1.672310],accel_mss,speed_ms,0,blend_radius_m)
    |   movel([0.101707, -1.432553, -2.528235, -0.751601, 1.570796, 1.672503],accel_mss,speed_ms,0,blend_radius_m)
    |   movel([0.101503, -1.431056, -2.529407, -0.751926, 1.570796, 1.672299],accel_mss,speed_ms,0,blend_radius_m)
    |   movel([0.100596, -1.429995, -2.530235, -0.752159, 1.570796, 1.671393],accel_mss,speed_ms,0,blend_radius_m)
    |   movel([0.099697, -1.429566, -2.530569, -0.752254, 1.570796, 1.670494],accel_mss,speed_ms,0,blend_radius_m)
    |   movel([0.098793, -1.429491, -2.530627, -0.752270, 1.570796, 1.669589],accel_mss,speed_ms,0,blend_radius_m)
    |   movel([0.097963, -1.429720, -2.530449, -0.752220, 1.570796, 1.668759],accel_mss,speed_ms,0,blend_radius_m)
    |   movel([0.097276, -1.430214, -2.530064, -0.752111, 1.570796, 1.668072],accel_mss,speed_ms,0,blend_radius_m)
    |   movel([0.096732, -1.431251, -2.529254, -0.751884, 1.570796, 1.667529],accel_mss,speed_ms,0,blend_radius_m)
    |   movel([0.096287, -1.432279, -2.528450, -0.751660, 1.570796, 1.667083],accel_mss,speed_ms,0,blend_radius_m)
    |   movel([0.095363, -1.433428, -2.527549, -0.751412, 1.570796, 1.666159],accel_mss,speed_ms,0,blend_radius_m)
    |   movel([0.093925, -1.434552, -2.526666, -0.751171, 1.570796, 1.664721],accel_mss,speed_ms,0,blend_radius_m)
    |   movel([0.092399, -1.435087, -2.526245, -0.751057, 1.570796, 1.663196],accel_mss,speed_ms,0,blend_radius_m)
    |   movel([0.090939, -1.435088, -2.526244, -0.751057, 1.570796, 1.661735],accel_mss,speed_ms,0,blend_radius_m)
    |   movel([0.089706, -1.434602, -2.526627, -0.751160, 1.570796, 1.660503],accel_mss,speed_ms,0,blend_radius_m)
    |   movel([0.088851, -1.433727, -2.527315, -0.751348, 1.570796, 1.659647],accel_mss,speed_ms,0,blend_radius_m)
    |   movel([0.088526, -1.432563, -2.528227, -0.751598, 1.570796, 1.659322],accel_mss,speed_ms,0,blend_radius_m)
    |   movel([0.088829, -1.431224, -2.529275, -0.751890, 1.570796, 1.659626],accel_mss,speed_ms,0,blend_radius_m)
    |   movel([0.089862, -1.429823, -2.530369, -0.752197, 1.570796, 1.660658],accel_mss,speed_ms,0,blend_radius_m)
    |   movel([0.091068, -1.428780, -2.531181, -0.752428, 1.570796, 1.661865],accel_mss,speed_ms,0,blend_radius_m)
    |   movel([0.092383, -1.428029, -2.531765, -0.752595, 1.570796, 1.663180],accel_mss,speed_ms,0,blend_radius_m)
    |   movel([0.093800, -1.427571, -2.532121, -0.752697, 1.570796, 1.664596],accel_mss,speed_ms,0,blend_radius_m)
    |   movel([0.095318, -1.427407, -2.532248, -0.752734, 1.570796, 1.666114],accel_mss,speed_ms,0,blend_radius_m)
    |   movel([0.096869, -1.427511, -2.532167, -0.752711, 1.570796, 1.667665],accel_mss,speed_ms,0,blend_radius_m)
    |   movel([0.098384, -1.427860, -2.531896, -0.752633, 1.570796, 1.669180],accel_mss,speed_ms,0,blend_radius_m)
    |   movel([0.101302, -1.429281, -2.530791, -0.752317, 1.570796, 1.672098],accel_mss,speed_ms,0,blend_radius_m)
    |   movel([0.102869, -1.430520, -2.529825, -0.752044, 1.570796, 1.673665],accel_mss,speed_ms,0,blend_radius_m)
    |   movel([0.104126, -1.431914, -2.528736, -0.751739, 1.570796, 1.674922],accel_mss,speed_ms,0,blend_radius_m)
    |   movel([0.105072, -1.433460, -2.527524, -0.751405, 1.570796, 1.675868],accel_mss,speed_ms,0,blend_radius_m)
    |   movel([0.105708, -1.435158, -2.526189, -0.751042, 1.570796, 1.676504],accel_mss,speed_ms,0,blend_radius_m)
    |   movel([0.105875, -1.436962, -2.524766, -0.750661, 1.570796, 1.676672],accel_mss,speed_ms,0,blend_radius_m)
    |   movel([0.105413, -1.438830, -2.523287, -0.750272, 1.570796, 1.676209],accel_mss,speed_ms,0,blend_radius_m)
    |   movel([0.104327, -1.440758, -2.521755, -0.749876, 1.570796, 1.675124],accel_mss,speed_ms,0,blend_radius_m)
    |   movel([0.102618, -1.442749, -2.520167, -0.749473, 1.570796, 1.673414],accel_mss,speed_ms,0,blend_radius_m)
    |   movel([0.100753, -1.444369, -2.518871, -0.749149, 1.570796, 1.671549],accel_mss,speed_ms,0,blend_radius_m)
    |   movel([0.098712, -1.445664, -2.517832, -0.748893, 1.570796, 1.669508],accel_mss,speed_ms,0,blend_radius_m)
    |   movel([0.096580, -1.446682, -2.517013, -0.748694, 1.570796, 1.667376],accel_mss,speed_ms,0,blend_radius_m)
    |   movel([0.094453, -1.447465, -2.516382, -0.748542, 1.570796, 1.665249],accel_mss,speed_ms,0,blend_radius_m)
    |   movel([0.089204, -1.448866, -2.515251, -0.748272, 1.570796, 1.660000],accel_mss,speed_ms,0,blend_radius_m)
    |   movel([0.084253, -1.450226, -2.514150, -0.748013, 1.570796, 1.655049],accel_mss,speed_ms,0,blend_radius_m)
    |   movel([0.082323, -1.450941, -2.513570, -0.747877, 1.570796, 1.653120],accel_mss,speed_ms,0,blend_radius_m)
    |   movel([0.080426, -1.451855, -2.512828, -0.747706, 1.570796, 1.651222],accel_mss,speed_ms,0,blend_radius_m)
    |   movel([0.078646, -1.452992, -2.511903, -0.747494, 1.570796, 1.649443],accel_mss,speed_ms,0,blend_radius_m)
    |   movel([0.077077, -1.454379, -2.510772, -0.747238, 1.570796, 1.647873],accel_mss,speed_ms,0,blend_radius_m)
    |   movel([0.077721, -1.454788, -2.510438, -0.747163, 1.570796, 1.648517],accel_mss,speed_ms,0,blend_radius_m)
    |   movel([0.079611, -1.455815, -2.509597, -0.746977, 1.570796, 1.650407],accel_mss,speed_ms,0,blend_radius_m)
    |   movel([0.081484, -1.456496, -2.509039, -0.746854, 1.570796, 1.652280],accel_mss,speed_ms,0,blend_radius_m)
    |   movel([0.083340, -1.456829, -2.508766, -0.746794, 1.570796, 1.654136],accel_mss,speed_ms,0,blend_radius_m)
    |   movel([0.085185, -1.456812, -2.508780, -0.746797, 1.570796, 1.655981],accel_mss,speed_ms,0,blend_radius_m)
    |   movel([0.086996, -1.456490, -2.509044, -0.746855, 1.570796, 1.657792],accel_mss,speed_ms,0,blend_radius_m)
    |   movel([0.088744, -1.455908, -2.509521, -0.746960, 1.570796, 1.659540],accel_mss,speed_ms,0,blend_radius_m)
    |   movel([0.090437, -1.455062, -2.510213, -0.747113, 1.570796, 1.661233],accel_mss,speed_ms,0,blend_radius_m)
    |   movel([0.092073, -1.453953, -2.511120, -0.747317, 1.570796, 1.662869],accel_mss,speed_ms,0,blend_radius_m)
    |   movel([0.085333, -1.460787, -2.505507, -0.746096, 1.570796, 1.656129],accel_mss,speed_ms,0,blend_radius_m)
    |   movel([0.068092, -1.449897, -2.514417, -0.748075, 1.570796, 1.638889],accel_mss,speed_ms,0,blend_radius_m)
    |   movel([0.068760, -1.449197, -2.514984, -0.748208, 1.570796, 1.639556],accel_mss,speed_ms,0,blend_radius_m)
    |   speed_ms = 0.003
    |   movel([0.068760, -1.443093, -2.512190, -0.757106, 1.570796, 1.639556],accel_mss,speed_ms,0,blend_radius_m)
    |   speed_ms = 0.05
    |   movel([0.068760, -1.419496, -2.500728, -0.792166, 1.570796, 1.639556],accel_mss,speed_ms,0,blend_radius_m)
    |   #M_RunCode9
    |   movel([0.091644, -1.428444, -2.493753, -0.790192, 1.570796, 1.662440],accel_mss,speed_ms,0,blend_radius_m)
    |   #M_RunCode3
    |   movel([0.091644, -1.451861, -2.505107, -0.755421, 1.570796, 1.662440],accel_mss,speed_ms,0,blend_radius_m)
    |   speed_ms = 0.003
    |   movel([0.091644, -1.457915, -2.507874, -0.746600, 1.570796, 1.662440],accel_mss,speed_ms,0,blend_radius_m)
    |   speed_ms = 0.02
    |   movel([0.093047, -1.456830, -2.508765, -0.746794, 1.570796, 1.663844],accel_mss,speed_ms,0,blend_radius_m)
    |   movel([0.094548, -1.456307, -2.509194, -0.746888, 1.570796, 1.665344],accel_mss,speed_ms,0,blend_radius_m)
    |   movel([0.095984, -1.456307, -2.509194, -0.746888, 1.570796, 1.666781],accel_mss,speed_ms,0,blend_radius_m)
    |   movel([0.097185, -1.456794, -2.508795, -0.746800, 1.570796, 1.667982],accel_mss,speed_ms,0,blend_radius_m)
    |   movel([0.098001, -1.457663, -2.508081, -0.746645, 1.570796, 1.668797],accel_mss,speed_ms,0,blend_radius_m)
    |   movel([0.098284, -1.458816, -2.507133, -0.746440, 1.570796, 1.669081],accel_mss,speed_ms,0,blend_radius_m)
    |   movel([0.097962, -1.460123, -2.506055, -0.746211, 1.570796, 1.668759],accel_mss,speed_ms,0,blend_radius_m)
    |   movel([0.096952, -1.461458, -2.504951, -0.745979, 1.570796, 1.667749],accel_mss,speed_ms,0,blend_radius_m)
    |   movel([0.095818, -1.462389, -2.504180, -0.745820, 1.570796, 1.666614],accel_mss,speed_ms,0,blend_radius_m)
    |   movel([0.094731, -1.462927, -2.503734, -0.745728, 1.570796, 1.665527],accel_mss,speed_ms,0,blend_radius_m)
    |   movel([0.093654, -1.463543, -2.503222, -0.745623, 1.570796, 1.664451],accel_mss,speed_ms,0,blend_radius_m)
    |   movel([0.093235, -1.464167, -2.502704, -0.745518, 1.570796, 1.664031],accel_mss,speed_ms,0,blend_radius_m)
    |   movel([0.093155, -1.464858, -2.502129, -0.745402, 1.570796, 1.663951],accel_mss,speed_ms,0,blend_radius_m)
    |   movel([0.093385, -1.465511, -2.501584, -0.745293, 1.570796, 1.664181],accel_mss,speed_ms,0,blend_radius_m)
    |   movel([0.093901, -1.466023, -2.501158, -0.745209, 1.570796, 1.664698],accel_mss,speed_ms,0,blend_radius_m)
    |   movel([0.094816, -1.466465, -2.500788, -0.745136, 1.570796, 1.665612],accel_mss,speed_ms,0,blend_radius_m)
    |   movel([0.095859, -1.466661, -2.500625, -0.745103, 1.570796, 1.666655],accel_mss,speed_ms,0,blend_radius_m)
    |   movel([0.097030, -1.466609, -2.500669, -0.745112, 1.570796, 1.667826],accel_mss,speed_ms,0,blend_radius_m)
    |   movel([0.098335, -1.466306, -2.500921, -0.745162, 1.570796, 1.669131],accel_mss,speed_ms,0,blend_radius_m)
    |   movel([0.099693, -1.465776, -2.501364, -0.745249, 1.570796, 1.670489],accel_mss,speed_ms,0,blend_radius_m)
    |   movel([0.101031, -1.465031, -2.501985, -0.745373, 1.570796, 1.671828],accel_mss,speed_ms,0,blend_radius_m)
    |   movel([0.102349, -1.464074, -2.502781, -0.745534, 1.570796, 1.673146],accel_mss,speed_ms,0,blend_radius_m)
    |   movel([0.103652, -1.462901, -2.503755, -0.745732, 1.570796, 1.674448],accel_mss,speed_ms,0,blend_radius_m)
    |   movel([0.105460, -1.460691, -2.505586, -0.746112, 1.570796, 1.676256],accel_mss,speed_ms,0,blend_radius_m)
    |   movel([0.106567, -1.458339, -2.507526, -0.746525, 1.570796, 1.677363],accel_mss,speed_ms,0,blend_radius_m)
    |   movel([0.106833, -1.457125, -2.508524, -0.746741, 1.570796, 1.677629],accel_mss,speed_ms,0,blend_radius_m)
    |   movel([0.106875, -1.455909, -2.509520, -0.746960, 1.570796, 1.677671],accel_mss,speed_ms,0,blend_radius_m)
    |   movel([0.106293, -1.453467, -2.511516, -0.747406, 1.570796, 1.677089],accel_mss,speed_ms,0,blend_radius_m)
    |   movel([0.104760, -1.451110, -2.513434, -0.747846, 1.570796, 1.675557],accel_mss,speed_ms,0,blend_radius_m)
    |   movel([0.102219, -1.448940, -2.515191, -0.748258, 1.570796, 1.673015],accel_mss,speed_ms,0,blend_radius_m)
    |   movel([0.112879, -1.438335, -2.523679, -0.750375, 1.570796, 1.683675],accel_mss,speed_ms,0,blend_radius_m)
    |   movel([0.125357, -1.447246, -2.516558, -0.748584, 1.570796, 1.696153],accel_mss,speed_ms,0,blend_radius_m)
    |   movel([0.118375, -1.454033, -2.511054, -0.747302, 1.570796, 1.689171],accel_mss,speed_ms,0,blend_radius_m)
    |   movel([0.119565, -1.452078, -2.512647, -0.747664, 1.570796, 1.690361],accel_mss,speed_ms,0,blend_radius_m)
    |   movel([0.120216, -1.449982, -2.514348, -0.748059, 1.570796, 1.691012],accel_mss,speed_ms,0,blend_radius_m)
    |   movel([0.120286, -1.447853, -2.516069, -0.748467, 1.570796, 1.691082],accel_mss,speed_ms,0,blend_radius_m)
    |   movel([0.119744, -1.445795, -2.517726, -0.748868, 1.570796, 1.690540],accel_mss,speed_ms,0,blend_radius_m)
    |   movel([0.118574, -1.443902, -2.519245, -0.749242, 1.570796, 1.689371],accel_mss,speed_ms,0,blend_radius_m)
    |   movel([0.116776, -1.442270, -2.520550, -0.749569, 1.570796, 1.687572],accel_mss,speed_ms,0,blend_radius_m)
    |   movel([0.108891, -1.450046, -2.514296, -0.748047, 1.570796, 1.679687],accel_mss,speed_ms,0,blend_radius_m)
    |   movel([0.111149, -1.451987, -2.512721, -0.747681, 1.570796, 1.681946],accel_mss,speed_ms,0,blend_radius_m)
    |   movel([0.112862, -1.454281, -2.510852, -0.747256, 1.570796, 1.683658],accel_mss,speed_ms,0,blend_radius_m)
    |   movel([0.113843, -1.456836, -2.508760, -0.746793, 1.570796, 1.684640],accel_mss,speed_ms,0,blend_radius_m)
    |   movel([0.113996, -1.458177, -2.507659, -0.746553, 1.570796, 1.684792],accel_mss,speed_ms,0,blend_radius_m)
    |   movel([0.113921, -1.459562, -2.506518, -0.746309, 1.570796, 1.684717],accel_mss,speed_ms,0,blend_radius_m)
    |   movel([0.113584, -1.460961, -2.505363, -0.746065, 1.570796, 1.684380],accel_mss,speed_ms,0,blend_radius_m)
    |   movel([0.112946, -1.462346, -2.504216, -0.745827, 1.570796, 1.683742],accel_mss,speed_ms,0,blend_radius_m)
    |   movel([0.112010, -1.463719, -2.503077, -0.745594, 1.570796, 1.682807],accel_mss,speed_ms,0,blend_radius_m)
    |   movel([0.110776, -1.465079, -2.501945, -0.745365, 1.570796, 1.681573],accel_mss,speed_ms,0,blend_radius_m)
    |   movel([0.109370, -1.466315, -2.500914, -0.745160, 1.570796, 1.680166],accel_mss,speed_ms,0,blend_radius_m)
    |   movel([0.107913, -1.467322, -2.500072, -0.744995, 1.570796, 1.678709],accel_mss,speed_ms,0,blend_radius_m)
    |   movel([0.106405, -1.468100, -2.499420, -0.744868, 1.570796, 1.677201],accel_mss,speed_ms,0,blend_radius_m)
    |   movel([0.104842, -1.468651, -2.498959, -0.744779, 1.570796, 1.675639],accel_mss,speed_ms,0,blend_radius_m)
    |   movel([0.101726, -1.469166, -2.498526, -0.744696, 1.570796, 1.672522],accel_mss,speed_ms,0,blend_radius_m)
    |   movel([0.098732, -1.468965, -2.498695, -0.744729, 1.570796, 1.669529],accel_mss,speed_ms,0,blend_radius_m)
    |   movel([0.095976, -1.468176, -2.499357, -0.744856, 1.570796, 1.666772],accel_mss,speed_ms,0,blend_radius_m)
    |   movel([0.093579, -1.466926, -2.500403, -0.745060, 1.570796, 1.664375],accel_mss,speed_ms,0,blend_radius_m)
    |   movel([0.092215, -1.465786, -2.501355, -0.745248, 1.570796, 1.663012],accel_mss,speed_ms,0,blend_radius_m)
    |   movel([0.091101, -1.464365, -2.502539, -0.745485, 1.570796, 1.661898],accel_mss,speed_ms,0,blend_radius_m)
    |   movel([0.090369, -1.462764, -2.503870, -0.745756, 1.570796, 1.661165],accel_mss,speed_ms,0,blend_radius_m)
    |   movel([0.090161, -1.461082, -2.505263, -0.746044, 1.570796, 1.660957],accel_mss,speed_ms,0,blend_radius_m)
    |   movel([0.090557, -1.459431, -2.506626, -0.746332, 1.570796, 1.661353],accel_mss,speed_ms,0,blend_radius_m)
    |   movel([0.091644, -1.457915, -2.507874, -0.746600, 1.570796, 1.662440],accel_mss,speed_ms,0,blend_radius_m)
    |   speed_ms = 0.003
    |   movel([0.091644, -1.451861, -2.505107, -0.755421, 1.570796, 1.662440],accel_mss,speed_ms,0,blend_radius_m)
    |   speed_ms = 0.05
    |   movel([0.091644, -1.428444, -2.493753, -0.790192, 1.570796, 1.662440],accel_mss,speed_ms,0,blend_radius_m)
    |   #M_RunCode9
    |   movel([0.060488, -1.370560, -2.536857, -0.804973, 1.570796, 1.631284],accel_mss,speed_ms,0,blend_radius_m)
    |   #M_RunCode3
    |   movel([0.060488, -1.395107, -2.548924, -0.768359, 1.570796, 1.631284],accel_mss,speed_ms,0,blend_radius_m)
    |   speed_ms = 0.003
    |   movel([0.060488, -1.401474, -2.551869, -0.759046, 1.570796, 1.631284],accel_mss,speed_ms,0,blend_radius_m)
    |   speed_ms = 0.02
    |   movel([0.057912, -1.402882, -2.550829, -0.758678, 1.570796, 1.628708],accel_mss,speed_ms,0,blend_radius_m)
    |   movel([0.055150, -1.403883, -2.550088, -0.758418, 1.570796, 1.625946],accel_mss,speed_ms,0,blend_radius_m)
    |   movel([0.052304, -1.404524, -2.549612, -0.758252, 1.570796, 1.623100],accel_mss,speed_ms,0,blend_radius_m)
    |   movel([0.049478, -1.404845, -2.549374, -0.758170, 1.570796, 1.620274],accel_mss,speed_ms,0,blend_radius_m)
    |   movel([0.046779, -1.404883, -2.549346, -0.758160, 1.570796, 1.617575],accel_mss,speed_ms,0,blend_radius_m)
    |   movel([0.046830, -1.402197, -2.551335, -0.758857, 1.570796, 1.617627],accel_mss,speed_ms,0,blend_radius_m)
    |   movel([0.047701, -1.399025, -2.553670, -0.759694, 1.570796, 1.618497],accel_mss,speed_ms,0,blend_radius_m)
    |   movel([0.049282, -1.395655, -2.556135, -0.760599, 1.570796, 1.620078],accel_mss,speed_ms,0,blend_radius_m)
    |   movel([0.051452, -1.392398, -2.558502, -0.761489, 1.570796, 1.622248],accel_mss,speed_ms,0,blend_radius_m)
    |   movel([0.054094, -1.389561, -2.560551, -0.762277, 1.570796, 1.624891],accel_mss,speed_ms,0,blend_radius_m)
    |   movel([0.055551, -1.388400, -2.561386, -0.762603, 1.570796, 1.626347],accel_mss,speed_ms,0,blend_radius_m)
    |   movel([0.057075, -1.387463, -2.562058, -0.762868, 1.570796, 1.627871],accel_mss,speed_ms,0,blend_radius_m)
    |   movel([0.058652, -1.386791, -2.562540, -0.763058, 1.570796, 1.629448],accel_mss,speed_ms,0,blend_radius_m)
    |   movel([0.060264, -1.386424, -2.562802, -0.763162, 1.570796, 1.631060],accel_mss,speed_ms,0,blend_radius_m)
    |   movel([0.061891, -1.386400, -2.562820, -0.763169, 1.570796, 1.632687],accel_mss,speed_ms,0,blend_radius_m)
    |   movel([0.063514, -1.386763, -2.562560, -0.763066, 1.570796, 1.634311],accel_mss,speed_ms,0,blend_radius_m)
    |   movel([0.065406, -1.387920, -2.561731, -0.762739, 1.570796, 1.636202],accel_mss,speed_ms,0,blend_radius_m)
    |   movel([0.066409, -1.389653, -2.560484, -0.762252, 1.570796, 1.637205],accel_mss,speed_ms,0,blend_radius_m)
    |   movel([0.066594, -1.391847, -2.558900, -0.761641, 1.570796, 1.637391],accel_mss,speed_ms,0,blend_radius_m)
    |   movel([0.066032, -1.394384, -2.557060, -0.760944, 1.570796, 1.636828],accel_mss,speed_ms,0,blend_radius_m)
    |   movel([0.064655, -1.397272, -2.554954, -0.760162, 1.570796, 1.635452],accel_mss,speed_ms,0,blend_radius_m)
    |   movel([0.062771, -1.399619, -2.553234, -0.759536, 1.570796, 1.633568],accel_mss,speed_ms,0,blend_radius_m)
    |   movel([0.060488, -1.401474, -2.551869, -0.759046, 1.570796, 1.631284],accel_mss,speed_ms,0,blend_radius_m)
    |   speed_ms = 0.003
    |   movel([0.060488, -1.395107, -2.548924, -0.768359, 1.570796, 1.631284],accel_mss,speed_ms,0,blend_radius_m)
    |   speed_ms = 0.05
    |   movel([0.060488, -1.370560, -2.536857, -0.804973, 1.570796, 1.631284],accel_mss,speed_ms,0,blend_radius_m)
    |   #M_RunCode9
    |   movel([0.102810, -1.281657, -2.594206, -0.836526, 1.570796, 1.673607],accel_mss,speed_ms,0,blend_radius_m)
    |   #M_RunCode3
    |   movel([0.102810, -1.307703, -2.607417, -0.797270, 1.570796, 1.673607],accel_mss,speed_ms,0,blend_radius_m)
    |   speed_ms = 0.003
    |   movel([0.102810, -1.314498, -2.610649, -0.787241, 1.570796, 1.673607],accel_mss,speed_ms,0,blend_radius_m)
    |   speed_ms = 0.007
    |   movel([0.101124, -1.314285, -2.610781, -0.787324, 1.570796, 1.671920],accel_mss,speed_ms,0,blend_radius_m)
    |   movel([0.099693, -1.313627, -2.611185, -0.787576, 1.570796, 1.670490],accel_mss,speed_ms,0,blend_radius_m)
    |   movel([0.098422, -1.312733, -2.611735, -0.787921, 1.570796, 1.669218],accel_mss,speed_ms,0,blend_radius_m)
    |   movel([0.099152, -1.312243, -2.612036, -0.788110, 1.570796, 1.669948],accel_mss,speed_ms,0,blend_radius_m)
    |   movel([0.099808, -1.312246, -2.612034, -0.788109, 1.570796, 1.670605],accel_mss,speed_ms,0,blend_radius_m)
    |   movel([0.100590, -1.312198, -2.612063, -0.788128, 1.570796, 1.671386],accel_mss,speed_ms,0,blend_radius_m)
    |   movel([0.101690, -1.311561, -2.612454, -0.788374, 1.570796, 1.672486],accel_mss,speed_ms,0,blend_radius_m)
    |   movel([0.102667, -1.310546, -2.613075, -0.788768, 1.570796, 1.673464],accel_mss,speed_ms,0,blend_radius_m)
    |   movel([0.103478, -1.309414, -2.613765, -0.789209, 1.570796, 1.674274],accel_mss,speed_ms,0,blend_radius_m)
    |   movel([0.104551, -1.307819, -2.614737, -0.789834, 1.570796, 1.675348],accel_mss,speed_ms,0,blend_radius_m)
    |   movel([0.103059, -1.306582, -2.615487, -0.790320, 1.570796, 1.673855],accel_mss,speed_ms,0,blend_radius_m)
    |   movel([0.101322, -1.306101, -2.615778, -0.790510, 1.570796, 1.672118],accel_mss,speed_ms,0,blend_radius_m)
    |   movel([0.100360, -1.306234, -2.615698, -0.790457, 1.570796, 1.671156],accel_mss,speed_ms,0,blend_radius_m)
    |   movel([0.099335, -1.306666, -2.615436, -0.790287, 1.570796, 1.670132],accel_mss,speed_ms,0,blend_radius_m)
    |   movel([0.098248, -1.307435, -2.614970, -0.789985, 1.570796, 1.669044],accel_mss,speed_ms,0,blend_radius_m)
    |   movel([0.097100, -1.308574, -2.614277, -0.789538, 1.570796, 1.667896],accel_mss,speed_ms,0,blend_radius_m)
    |   movel([0.096912, -1.307374, -2.615007, -0.790008, 1.570796, 1.667709],accel_mss,speed_ms,0,blend_radius_m)
    |   movel([0.096937, -1.306264, -2.615679, -0.790445, 1.570796, 1.667734],accel_mss,speed_ms,0,blend_radius_m)
    |   movel([0.097128, -1.305794, -2.615964, -0.790631, 1.570796, 1.667925],accel_mss,speed_ms,0,blend_radius_m)
    |   movel([0.097494, -1.305410, -2.616196, -0.790783, 1.570796, 1.668290],accel_mss,speed_ms,0,blend_radius_m)
    |   movel([0.098903, -1.304980, -2.616456, -0.790953, 1.570796, 1.669699],accel_mss,speed_ms,0,blend_radius_m)
    |   movel([0.101602, -1.305034, -2.616424, -0.790932, 1.570796, 1.672398],accel_mss,speed_ms,0,blend_radius_m)
    |   movel([0.104000, -1.305726, -2.616005, -0.790658, 1.570796, 1.674796],accel_mss,speed_ms,0,blend_radius_m)
    |   movel([0.104911, -1.306348, -2.615629, -0.790412, 1.570796, 1.675707],accel_mss,speed_ms,0,blend_radius_m)
    |   movel([0.105534, -1.307180, -2.615125, -0.790085, 1.570796, 1.676331],accel_mss,speed_ms,0,blend_radius_m)
    |   movel([0.105803, -1.308230, -2.614487, -0.789673, 1.570796, 1.676600],accel_mss,speed_ms,0,blend_radius_m)
    |   movel([0.105647, -1.309515, -2.613704, -0.789170, 1.570796, 1.676443],accel_mss,speed_ms,0,blend_radius_m)
    |   movel([0.103926, -1.309531, -2.613694, -0.789164, 1.570796, 1.674722],accel_mss,speed_ms,0,blend_radius_m)
    |   movel([0.104851, -1.314057, -2.610921, -0.787411, 1.570796, 1.675647],accel_mss,speed_ms,0,blend_radius_m)
    |   movel([0.102810, -1.314498, -2.610649, -0.787241, 1.570796, 1.673607],accel_mss,speed_ms,0,blend_radius_m)
    |   speed_ms = 0.003
    |   movel([0.102810, -1.307703, -2.607417, -0.797270, 1.570796, 1.673607],accel_mss,speed_ms,0,blend_radius_m)
    |   speed_ms = 0.05
    |   movel([0.102810, -1.281657, -2.594206, -0.836526, 1.570796, 1.673607],accel_mss,speed_ms,0,blend_radius_m)
    |   #M_RunCode9
    |   movel([0.062673, -1.265901, -2.603322, -0.843166, 1.570796, 1.633469],accel_mss,speed_ms,0,blend_radius_m)
    |   #M_RunCode3
    |   movel([0.062673, -1.292173, -2.616738, -0.803478, 1.570796, 1.633469],accel_mss,speed_ms,0,blend_radius_m)
    |   speed_ms = 0.003
    |   movel([0.062673, -1.299035, -2.620023, -0.793331, 1.570796, 1.633469],accel_mss,speed_ms,0,blend_radius_m)
    |   speed_ms = 0.02
    |   movel([0.060971, -1.301295, -2.618672, -0.792422, 1.570796, 1.631768],accel_mss,speed_ms,0,blend_radius_m)
    |   movel([0.059037, -1.303474, -2.617364, -0.791551, 1.570796, 1.629833],accel_mss,speed_ms,0,blend_radius_m)
    |   movel([0.056880, -1.305538, -2.616119, -0.790732, 1.570796, 1.627676],accel_mss,speed_ms,0,blend_radius_m)
    |   movel([0.054516, -1.307458, -2.614956, -0.789975, 1.570796, 1.625312],accel_mss,speed_ms,0,blend_radius_m)
    |   movel([0.051966, -1.309202, -2.613895, -0.789292, 1.570796, 1.622762],accel_mss,speed_ms,0,blend_radius_m)
    |   movel([0.050531, -1.309908, -2.613464, -0.789017, 1.570796, 1.621327],accel_mss,speed_ms,0,blend_radius_m)
    |   movel([0.048992, -1.310471, -2.613121, -0.788798, 1.570796, 1.619788],accel_mss,speed_ms,0,blend_radius_m)
    |   movel([0.047608, -1.310986, -2.612806, -0.788597, 1.570796, 1.618404],accel_mss,speed_ms,0,blend_radius_m)
    |   movel([0.046652, -1.311534, -2.612470, -0.788385, 1.570796, 1.617448],accel_mss,speed_ms,0,blend_radius_m)
    |   movel([0.045483, -1.312989, -2.611578, -0.787822, 1.570796, 1.616280],accel_mss,speed_ms,0,blend_radius_m)
    |   movel([0.044130, -1.315113, -2.610270, -0.787006, 1.570796, 1.614926],accel_mss,speed_ms,0,blend_radius_m)
    |   movel([0.042745, -1.317335, -2.608896, -0.786158, 1.570796, 1.613542],accel_mss,speed_ms,0,blend_radius_m)
    |   movel([0.041473, -1.319096, -2.607802, -0.785491, 1.570796, 1.612270],accel_mss,speed_ms,0,blend_radius_m)
    |   movel([0.038551, -1.322121, -2.605913, -0.784355, 1.570796, 1.609348],accel_mss,speed_ms,0,blend_radius_m)
    |   movel([0.035652, -1.324487, -2.604427, -0.783475, 1.570796, 1.606448],accel_mss,speed_ms,0,blend_radius_m)
    |   movel([0.032775, -1.326262, -2.603308, -0.782820, 1.570796, 1.603571],accel_mss,speed_ms,0,blend_radius_m)
    |   movel([0.029921, -1.327506, -2.602520, -0.782363, 1.570796, 1.600718],accel_mss,speed_ms,0,blend_radius_m)
    |   movel([0.027098, -1.328280, -2.602030, -0.782080, 1.570796, 1.597894],accel_mss,speed_ms,0,blend_radius_m)
    |   movel([0.024310, -1.328639, -2.601801, -0.781948, 1.570796, 1.595106],accel_mss,speed_ms,0,blend_radius_m)
    |   movel([0.021561, -1.328641, -2.601800, -0.781948, 1.570796, 1.592357],accel_mss,speed_ms,0,blend_radius_m)
    |   movel([0.018855, -1.328342, -2.601990, -0.782057, 1.570796, 1.589651],accel_mss,speed_ms,0,blend_radius_m)
    |   movel([0.013608, -1.327062, -2.602802, -0.782526, 1.570796, 1.584405],accel_mss,speed_ms,0,blend_radius_m)
    |   movel([0.008640, -1.325228, -2.603960, -0.783201, 1.570796, 1.579436],accel_mss,speed_ms,0,blend_radius_m)
    |   movel([-0.000140, -1.321616, -2.606229, -0.784544, 1.570796, 1.570657],accel_mss,speed_ms,0,blend_radius_m)
    |   movel([-0.004320, -1.320469, -2.606946, -0.784974, 1.570796, 1.566476],accel_mss,speed_ms,0,blend_radius_m)
    |   movel([-0.009452, -1.319595, -2.607491, -0.785303, 1.570796, 1.561344],accel_mss,speed_ms,0,blend_radius_m)
    |   movel([-0.015283, -1.319073, -2.607816, -0.785500, 1.570796, 1.555514],accel_mss,speed_ms,0,blend_radius_m)
    |   movel([-0.021548, -1.318977, -2.607875, -0.785536, 1.570796, 1.549248],accel_mss,speed_ms,0,blend_radius_m)
    |   movel([-0.027979, -1.319376, -2.607627, -0.785386, 1.570796, 1.542817],accel_mss,speed_ms,0,blend_radius_m)
    |   movel([-0.034301, -1.320323, -2.607037, -0.785029, 1.570796, 1.536495],accel_mss,speed_ms,0,blend_radius_m)
    |   movel([-0.040235, -1.321867, -2.606072, -0.784450, 1.570796, 1.530561],accel_mss,speed_ms,0,blend_radius_m)
    |   movel([-0.042969, -1.322877, -2.605439, -0.784073, 1.570796, 1.527828],accel_mss,speed_ms,0,blend_radius_m)
    |   movel([-0.045502, -1.324050, -2.604702, -0.783637, 1.570796, 1.525295],accel_mss,speed_ms,0,blend_radius_m)
    |   movel([-0.048048, -1.325495, -2.603792, -0.783102, 1.570796, 1.522749],accel_mss,speed_ms,0,blend_radius_m)
    |   movel([-0.050940, -1.327387, -2.602596, -0.782406, 1.570796, 1.519856],accel_mss,speed_ms,0,blend_radius_m)
    |   movel([-0.053974, -1.329660, -2.601152, -0.781576, 1.570796, 1.516823],accel_mss,speed_ms,0,blend_radius_m)
    |   movel([-0.056949, -1.332244, -2.599503, -0.780642, 1.570796, 1.513848],accel_mss,speed_ms,0,blend_radius_m)
    |   movel([-0.059657, -1.335061, -2.597695, -0.779633, 1.570796, 1.511139],accel_mss,speed_ms,0,blend_radius_m)
    |   movel([-0.061909, -1.338046, -2.595768, -0.778576, 1.570796, 1.508888],accel_mss,speed_ms,0,blend_radius_m)
    |   movel([-0.063504, -1.341126, -2.593765, -0.777497, 1.570796, 1.507292],accel_mss,speed_ms,0,blend_radius_m)
    |   movel([-0.063999, -1.342680, -2.592751, -0.776958, 1.570796, 1.506798],accel_mss,speed_ms,0,blend_radius_m)
    |   movel([-0.064257, -1.344233, -2.591733, -0.776423, 1.570796, 1.506539],accel_mss,speed_ms,0,blend_radius_m)
    |   movel([-0.064091, -1.346436, -2.590284, -0.775669, 1.570796, 1.506706],accel_mss,speed_ms,0,blend_radius_m)
    |   movel([-0.063209, -1.348011, -2.589244, -0.775134, 1.570796, 1.507587],accel_mss,speed_ms,0,blend_radius_m)
    |   movel([-0.061697, -1.349027, -2.588571, -0.774791, 1.570796, 1.509100],accel_mss,speed_ms,0,blend_radius_m)
    |   movel([-0.059635, -1.349546, -2.588227, -0.774616, 1.570796, 1.511162],accel_mss,speed_ms,0,blend_radius_m)
    |   movel([-0.057103, -1.349631, -2.588170, -0.774588, 1.570796, 1.513693],accel_mss,speed_ms,0,blend_radius_m)
    |   movel([-0.054182, -1.349345, -2.588360, -0.774684, 1.570796, 1.516614],accel_mss,speed_ms,0,blend_radius_m)
    |   movel([-0.050947, -1.348746, -2.588757, -0.774886, 1.570796, 1.519849],accel_mss,speed_ms,0,blend_radius_m)
    |   movel([-0.047477, -1.347898, -2.589319, -0.775172, 1.570796, 1.523319],accel_mss,speed_ms,0,blend_radius_m)
    |   movel([-0.040154, -1.345684, -2.590779, -0.775926, 1.570796, 1.530642],accel_mss,speed_ms,0,blend_radius_m)
    |   movel([-0.032847, -1.343171, -2.592429, -0.776789, 1.570796, 1.537949],accel_mss,speed_ms,0,blend_radius_m)
    |   movel([-0.026213, -1.340819, -2.593966, -0.777605, 1.570796, 1.544584],accel_mss,speed_ms,0,blend_radius_m)
    |   movel([-0.020917, -1.339093, -2.595088, -0.778208, 1.570796, 1.549880],accel_mss,speed_ms,0,blend_radius_m)
    |   movel([-0.008098, -1.335388, -2.597485, -0.779517, 1.570796, 1.562698],accel_mss,speed_ms,0,blend_radius_m)
    |   movel([-0.001242, -1.333585, -2.598644, -0.780160, 1.570796, 1.569554],accel_mss,speed_ms,0,blend_radius_m)
    |   movel([0.004075, -1.332484, -2.599350, -0.780556, 1.570796, 1.574872],accel_mss,speed_ms,0,blend_radius_m)
    |   movel([0.006089, -1.332313, -2.599459, -0.780617, 1.570796, 1.576885],accel_mss,speed_ms,0,blend_radius_m)
    |   movel([0.007962, -1.332384, -2.599414, -0.780592, 1.570796, 1.578758],accel_mss,speed_ms,0,blend_radius_m)
    |   movel([0.011274, -1.333194, -2.598895, -0.780300, 1.570796, 1.582071],accel_mss,speed_ms,0,blend_radius_m)
    |   movel([0.014005, -1.334783, -2.597874, -0.779732, 1.570796, 1.584801],accel_mss,speed_ms,0,blend_radius_m)
    |   movel([0.016157, -1.337009, -2.596439, -0.778942, 1.570796, 1.586953],accel_mss,speed_ms,0,blend_radius_m)
    |   movel([0.017725, -1.339735, -2.594671, -0.777983, 1.570796, 1.588521],accel_mss,speed_ms,0,blend_radius_m)
    |   movel([0.018714, -1.342828, -2.592654, -0.776907, 1.570796, 1.589510],accel_mss,speed_ms,0,blend_radius_m)
    |   movel([0.019132, -1.346151, -2.590472, -0.775766, 1.570796, 1.589928],accel_mss,speed_ms,0,blend_radius_m)
    |   movel([0.018983, -1.349568, -2.588212, -0.774609, 1.570796, 1.589779],accel_mss,speed_ms,0,blend_radius_m)
    |   movel([0.018040, -1.353888, -2.585332, -0.773169, 1.570796, 1.588836],accel_mss,speed_ms,0,blend_radius_m)
    |   movel([0.017330, -1.355729, -2.584097, -0.772563, 1.570796, 1.588126],accel_mss,speed_ms,0,blend_radius_m)
    |   movel([0.016466, -1.357392, -2.582978, -0.772019, 1.570796, 1.587262],accel_mss,speed_ms,0,blend_radius_m)
    |   movel([0.015462, -1.358898, -2.581961, -0.771531, 1.570796, 1.586259],accel_mss,speed_ms,0,blend_radius_m)
    |   movel([0.014321, -1.360271, -2.581030, -0.771088, 1.570796, 1.585118],accel_mss,speed_ms,0,blend_radius_m)
    |   movel([0.011664, -1.362722, -2.579363, -0.770304, 1.570796, 1.582460],accel_mss,speed_ms,0,blend_radius_m)
    |   movel([0.008551, -1.364931, -2.577853, -0.769605, 1.570796, 1.579347],accel_mss,speed_ms,0,blend_radius_m)
    |   movel([0.005045, -1.367086, -2.576374, -0.768929, 1.570796, 1.575842],accel_mss,speed_ms,0,blend_radius_m)
    |   movel([-0.002899, -1.371950, -2.573010, -0.767429, 1.570796, 1.567897],accel_mss,speed_ms,0,blend_radius_m)
    |   movel([-0.003291, -1.372227, -2.572817, -0.767344, 1.570796, 1.567506],accel_mss,speed_ms,0,blend_radius_m)
    |   movel([-0.003098, -1.372226, -2.572818, -0.767345, 1.570796, 1.567698],accel_mss,speed_ms,0,blend_radius_m)
    |   movel([-0.001268, -1.371533, -2.573300, -0.767556, 1.570796, 1.569529],accel_mss,speed_ms,0,blend_radius_m)
    |   movel([0.006076, -1.368405, -2.575465, -0.768519, 1.570796, 1.576872],accel_mss,speed_ms,0,blend_radius_m)
    |   movel([0.018333, -1.363222, -2.579022, -0.770145, 1.570796, 1.589129],accel_mss,speed_ms,0,blend_radius_m)
    |   movel([0.012601, -1.368195, -2.575610, -0.768584, 1.570796, 1.583397],accel_mss,speed_ms,0,blend_radius_m)
    |   movel([0.006067, -1.373477, -2.571947, -0.766964, 1.570796, 1.576863],accel_mss,speed_ms,0,blend_radius_m)
    |   movel([-0.000996, -1.378907, -2.568141, -0.765341, 1.570796, 1.569801],accel_mss,speed_ms,0,blend_radius_m)
    |   movel([-0.008330, -1.384316, -2.564308, -0.763765, 1.570796, 1.562466],accel_mss,speed_ms,0,blend_radius_m)
    |   movel([-0.022815, -1.394452, -2.557011, -0.760926, 1.570796, 1.547982],accel_mss,speed_ms,0,blend_radius_m)
    |   movel([-0.029489, -1.398858, -2.553793, -0.759738, 1.570796, 1.541307],accel_mss,speed_ms,0,blend_radius_m)
    |   movel([-0.035482, -1.402621, -2.551022, -0.758746, 1.570796, 1.535314],accel_mss,speed_ms,0,blend_radius_m)
    |   movel([-0.042163, -1.410108, -2.545446, -0.756834, 1.570796, 1.528633],accel_mss,speed_ms,0,blend_radius_m)
    |   movel([-0.048670, -1.417962, -2.539510, -0.754918, 1.570796, 1.522126],accel_mss,speed_ms,0,blend_radius_m)
    |   movel([-0.061315, -1.434043, -2.527066, -0.751280, 1.570796, 1.509481],accel_mss,speed_ms,0,blend_radius_m)
    |   movel([-0.067546, -1.441940, -2.520813, -0.749636, 1.570796, 1.503251],accel_mss,speed_ms,0,blend_radius_m)
    |   movel([-0.073784, -1.449537, -2.514708, -0.748144, 1.570796, 1.497012],accel_mss,speed_ms,0,blend_radius_m)
    |   movel([-0.080081, -1.456689, -2.508881, -0.746819, 1.570796, 1.490715],accel_mss,speed_ms,0,blend_radius_m)
    |   movel([-0.086500, -1.463258, -2.503460, -0.745672, 1.570796, 1.484296],accel_mss,speed_ms,0,blend_radius_m)
    |   movel([-0.089113, -1.465618, -2.501495, -0.745276, 1.570796, 1.481683],accel_mss,speed_ms,0,blend_radius_m)
    |   movel([-0.091712, -1.467683, -2.499770, -0.744936, 1.570796, 1.479084],accel_mss,speed_ms,0,blend_radius_m)
    |   movel([-0.094276, -1.469447, -2.498291, -0.744651, 1.570796, 1.476521],accel_mss,speed_ms,0,blend_radius_m)
    |   movel([-0.096785, -1.470911, -2.497060, -0.744419, 1.570796, 1.474011],accel_mss,speed_ms,0,blend_radius_m)
    |   movel([-0.099225, -1.472066, -2.496085, -0.744237, 1.570796, 1.471572],accel_mss,speed_ms,0,blend_radius_m)
    |   movel([-0.101576, -1.472911, -2.495372, -0.744106, 1.570796, 1.469221],accel_mss,speed_ms,0,blend_radius_m)
    |   movel([-0.103820, -1.473442, -2.494923, -0.744024, 1.570796, 1.466976],accel_mss,speed_ms,0,blend_radius_m)
    |   movel([-0.105937, -1.473654, -2.494744, -0.743992, 1.570796, 1.464859],accel_mss,speed_ms,0,blend_radius_m)
    |   movel([-0.107910, -1.473539, -2.494841, -0.744009, 1.570796, 1.462887],accel_mss,speed_ms,0,blend_radius_m)
    |   movel([-0.109720, -1.473091, -2.495220, -0.744078, 1.570796, 1.461076],accel_mss,speed_ms,0,blend_radius_m)
    |   movel([-0.111344, -1.472304, -2.495885, -0.744200, 1.570796, 1.459452],accel_mss,speed_ms,0,blend_radius_m)
    |   movel([-0.112768, -1.471173, -2.496839, -0.744377, 1.570796, 1.458028],accel_mss,speed_ms,0,blend_radius_m)
    |   movel([-0.113968, -1.469686, -2.498090, -0.744613, 1.570796, 1.456829],accel_mss,speed_ms,0,blend_radius_m)
    |   movel([-0.114922, -1.467834, -2.499643, -0.744912, 1.570796, 1.455875],accel_mss,speed_ms,0,blend_radius_m)
    |   movel([-0.115609, -1.465610, -2.501502, -0.745277, 1.570796, 1.455187],accel_mss,speed_ms,0,blend_radius_m)
    |   movel([-0.116006, -1.463000, -2.503674, -0.745715, 1.570796, 1.454790],accel_mss,speed_ms,0,blend_radius_m)
    |   movel([-0.112936, -1.462764, -2.503869, -0.745756, 1.570796, 1.457860],accel_mss,speed_ms,0,blend_radius_m)
    |   movel([-0.111418, -1.462572, -2.504029, -0.745788, 1.570796, 1.459378],accel_mss,speed_ms,0,blend_radius_m)
    |   movel([-0.109924, -1.462088, -2.504430, -0.745871, 1.570796, 1.460872],accel_mss,speed_ms,0,blend_radius_m)
    |   movel([-0.108807, -1.461396, -2.505003, -0.745990, 1.570796, 1.461989],accel_mss,speed_ms,0,blend_radius_m)
    |   movel([-0.107556, -1.460330, -2.505884, -0.746175, 1.570796, 1.463241],accel_mss,speed_ms,0,blend_radius_m)
    |   movel([-0.104733, -1.457261, -2.508412, -0.746717, 1.570796, 1.466063],accel_mss,speed_ms,0,blend_radius_m)
    |   movel([-0.101611, -1.453252, -2.511691, -0.747446, 1.570796, 1.469185],accel_mss,speed_ms,0,blend_radius_m)
    |   movel([-0.098360, -1.448678, -2.515403, -0.748308, 1.570796, 1.472436],accel_mss,speed_ms,0,blend_radius_m)
    |   movel([-0.092173, -1.439398, -2.522836, -0.750155, 1.570796, 1.478623],accel_mss,speed_ms,0,blend_radius_m)
    |   movel([-0.087668, -1.432622, -2.528181, -0.751586, 1.570796, 1.483129],accel_mss,speed_ms,0,blend_radius_m)
    |   movel([-0.083332, -1.426923, -2.532623, -0.752843, 1.570796, 1.487464],accel_mss,speed_ms,0,blend_radius_m)
    |   movel([-0.078941, -1.421179, -2.537051, -0.754159, 1.570796, 1.491855],accel_mss,speed_ms,0,blend_radius_m)
    |   movel([-0.091400, -1.427836, -2.531915, -0.752638, 1.570796, 1.479397],accel_mss,speed_ms,0,blend_radius_m)
    |   movel([-0.097928, -1.431068, -2.529397, -0.751924, 1.570796, 1.472868],accel_mss,speed_ms,0,blend_radius_m)
    |   movel([-0.104381, -1.433755, -2.527293, -0.751342, 1.570796, 1.466415],accel_mss,speed_ms,0,blend_radius_m)
    |   movel([-0.107519, -1.434780, -2.526486, -0.751122, 1.570796, 1.463277],accel_mss,speed_ms,0,blend_radius_m)
    |   movel([-0.110566, -1.435536, -2.525891, -0.750962, 1.570796, 1.460230],accel_mss,speed_ms,0,blend_radius_m)
    |   movel([-0.113501, -1.435974, -2.525546, -0.750869, 1.570796, 1.457296],accel_mss,speed_ms,0,blend_radius_m)
    |   movel([-0.116300, -1.436052, -2.525484, -0.750853, 1.570796, 1.454497],accel_mss,speed_ms,0,blend_radius_m)
    |   movel([-0.118941, -1.435725, -2.525742, -0.750922, 1.570796, 1.451855],accel_mss,speed_ms,0,blend_radius_m)
    |   movel([-0.121404, -1.434945, -2.526356, -0.751087, 1.570796, 1.449392],accel_mss,speed_ms,0,blend_radius_m)
    |   movel([-0.123665, -1.433664, -2.527364, -0.751361, 1.570796, 1.447131],accel_mss,speed_ms,0,blend_radius_m)
    |   movel([-0.125701, -1.431833, -2.528799, -0.751757, 1.570796, 1.445095],accel_mss,speed_ms,0,blend_radius_m)
    |   movel([-0.127479, -1.429180, -2.530870, -0.752339, 1.570796, 1.443317],accel_mss,speed_ms,0,blend_radius_m)
    |   movel([-0.128567, -1.425999, -2.533339, -0.753051, 1.570796, 1.442229],accel_mss,speed_ms,0,blend_radius_m)
    |   movel([-0.128974, -1.422404, -2.536111, -0.753874, 1.570796, 1.441823],accel_mss,speed_ms,0,blend_radius_m)
    |   movel([-0.128700, -1.418509, -2.539092, -0.754787, 1.570796, 1.442097],accel_mss,speed_ms,0,blend_radius_m)
    |   movel([-0.127750, -1.414438, -2.542185, -0.755766, 1.570796, 1.443046],accel_mss,speed_ms,0,blend_radius_m)
    |   movel([-0.126130, -1.410311, -2.545294, -0.756784, 1.570796, 1.444666],accel_mss,speed_ms,0,blend_radius_m)
    |   movel([-0.123845, -1.406255, -2.548326, -0.757808, 1.570796, 1.446951],accel_mss,speed_ms,0,blend_radius_m)
    |   movel([-0.120902, -1.402407, -2.551180, -0.758802, 1.570796, 1.449894],accel_mss,speed_ms,0,blend_radius_m)
    |   movel([-0.118903, -1.400597, -2.552515, -0.759277, 1.570796, 1.451893],accel_mss,speed_ms,0,blend_radius_m)
    |   movel([-0.116399, -1.398924, -2.553745, -0.759721, 1.570796, 1.454398],accel_mss,speed_ms,0,blend_radius_m)
    |   movel([-0.114170, -1.397957, -2.554453, -0.759979, 1.570796, 1.456626],accel_mss,speed_ms,0,blend_radius_m)
    |   movel([-0.113404, -1.397916, -2.554483, -0.759990, 1.570796, 1.457393],accel_mss,speed_ms,0,blend_radius_m)
    |   movel([-0.113001, -1.398265, -2.554228, -0.759896, 1.570796, 1.457795],accel_mss,speed_ms,0,blend_radius_m)
    |   movel([-0.114998, -1.399565, -2.553273, -0.759550, 1.570796, 1.455798],accel_mss,speed_ms,0,blend_radius_m)
    |   movel([-0.116593, -1.400819, -2.552351, -0.759219, 1.570796, 1.454203],accel_mss,speed_ms,0,blend_radius_m)
    |   movel([-0.117810, -1.402019, -2.551466, -0.758904, 1.570796, 1.452986],accel_mss,speed_ms,0,blend_radius_m)
    |   movel([-0.118672, -1.403156, -2.550626, -0.758607, 1.570796, 1.452124],accel_mss,speed_ms,0,blend_radius_m)
    |   movel([-0.119199, -1.404223, -2.549836, -0.758330, 1.570796, 1.451597],accel_mss,speed_ms,0,blend_radius_m)
    |   movel([-0.119413, -1.405206, -2.549106, -0.758077, 1.570796, 1.451383],accel_mss,speed_ms,0,blend_radius_m)
    |   movel([-0.119335, -1.406102, -2.548440, -0.757847, 1.570796, 1.451461],accel_mss,speed_ms,0,blend_radius_m)
    |   movel([-0.118989, -1.406902, -2.547844, -0.757643, 1.570796, 1.451807],accel_mss,speed_ms,0,blend_radius_m)
    |   movel([-0.117576, -1.408183, -2.546888, -0.757318, 1.570796, 1.453220],accel_mss,speed_ms,0,blend_radius_m)
    |   movel([-0.115345, -1.408986, -2.546287, -0.757116, 1.570796, 1.455451],accel_mss,speed_ms,0,blend_radius_m)
    |   movel([-0.112459, -1.409248, -2.546091, -0.757050, 1.570796, 1.458337],accel_mss,speed_ms,0,blend_radius_m)
    |   movel([-0.109083, -1.408906, -2.546347, -0.757136, 1.570796, 1.461714],accel_mss,speed_ms,0,blend_radius_m)
    |   movel([-0.106965, -1.408357, -2.546758, -0.757274, 1.570796, 1.463831],accel_mss,speed_ms,0,blend_radius_m)
    |   movel([-0.104406, -1.407446, -2.547439, -0.757505, 1.570796, 1.466390],accel_mss,speed_ms,0,blend_radius_m)
    |   movel([-0.098196, -1.404704, -2.549479, -0.758206, 1.570796, 1.472600],accel_mss,speed_ms,0,blend_radius_m)
    |   movel([-0.090922, -1.401036, -2.552191, -0.759162, 1.570796, 1.479874],accel_mss,speed_ms,0,blend_radius_m)
    |   movel([-0.083063, -1.396788, -2.555308, -0.760293, 1.570796, 1.487734],accel_mss,speed_ms,0,blend_radius_m)
    |   movel([-0.067573, -1.387951, -2.561708, -0.762730, 1.570796, 1.503223],accel_mss,speed_ms,0,blend_radius_m)
    |   movel([-0.055874, -1.381000, -2.566663, -0.764726, 1.570796, 1.514922],accel_mss,speed_ms,0,blend_radius_m)
    |   movel([-0.049959, -1.377461, -2.569159, -0.765769, 1.570796, 1.520837],accel_mss,speed_ms,0,blend_radius_m)
    |   movel([-0.046803, -1.375466, -2.570558, -0.766365, 1.570796, 1.523993],accel_mss,speed_ms,0,blend_radius_m)
    |   movel([-0.044493, -1.373787, -2.571731, -0.766871, 1.570796, 1.526303],accel_mss,speed_ms,0,blend_radius_m)
    |   movel([-0.043931, -1.373226, -2.572122, -0.767041, 1.570796, 1.526866],accel_mss,speed_ms,0,blend_radius_m)
    |   movel([-0.043801, -1.372867, -2.572373, -0.767150, 1.570796, 1.526996],accel_mss,speed_ms,0,blend_radius_m)
    |   movel([-0.044572, -1.372479, -2.572643, -0.767268, 1.570796, 1.526224],accel_mss,speed_ms,0,blend_radius_m)
    |   movel([-0.047476, -1.372220, -2.572823, -0.767346, 1.570796, 1.523320],accel_mss,speed_ms,0,blend_radius_m)
    |   movel([-0.050727, -1.372474, -2.572646, -0.767269, 1.570796, 1.520069],accel_mss,speed_ms,0,blend_radius_m)
    |   movel([-0.057799, -1.373319, -2.572057, -0.767012, 1.570796, 1.512998],accel_mss,speed_ms,0,blend_radius_m)
    |   movel([-0.061398, -1.373317, -2.572059, -0.767013, 1.570796, 1.509398],accel_mss,speed_ms,0,blend_radius_m)
    |   movel([-0.064898, -1.372629, -2.572538, -0.767222, 1.570796, 1.505898],accel_mss,speed_ms,0,blend_radius_m)
    |   movel([-0.066577, -1.371935, -2.573021, -0.767433, 1.570796, 1.504219],accel_mss,speed_ms,0,blend_radius_m)
    |   movel([-0.068195, -1.370958, -2.573699, -0.767732, 1.570796, 1.502601],accel_mss,speed_ms,0,blend_radius_m)
    |   movel([-0.069739, -1.369658, -2.574600, -0.768132, 1.570796, 1.501057],accel_mss,speed_ms,0,blend_radius_m)
    |   movel([-0.071195, -1.367994, -2.575748, -0.768647, 1.570796, 1.499601],accel_mss,speed_ms,0,blend_radius_m)
    |   movel([-0.072638, -1.365440, -2.577504, -0.769445, 1.570796, 1.498158],accel_mss,speed_ms,0,blend_radius_m)
    |   movel([-0.073373, -1.362616, -2.579435, -0.770338, 1.570796, 1.497424],accel_mss,speed_ms,0,blend_radius_m)
    |   movel([-0.073471, -1.359553, -2.581517, -0.771319, 1.570796, 1.497325],accel_mss,speed_ms,0,blend_radius_m)
    |   movel([-0.073008, -1.356295, -2.583717, -0.772377, 1.570796, 1.497789],accel_mss,speed_ms,0,blend_radius_m)
    |   movel([-0.072060, -1.352877, -2.586009, -0.773503, 1.570796, 1.498736],accel_mss,speed_ms,0,blend_radius_m)
    |   movel([-0.070704, -1.349346, -2.588360, -0.774684, 1.570796, 1.500092],accel_mss,speed_ms,0,blend_radius_m)
    |   movel([-0.069018, -1.345740, -2.590742, -0.775907, 1.570796, 1.501778],accel_mss,speed_ms,0,blend_radius_m)
    |   movel([-0.067084, -1.342109, -2.593124, -0.777156, 1.570796, 1.503712],accel_mss,speed_ms,0,blend_radius_m)
    |   movel([-0.062875, -1.335380, -2.597489, -0.779519, 1.570796, 1.507922],accel_mss,speed_ms,0,blend_radius_m)
    |   movel([-0.058564, -1.329688, -2.601135, -0.781566, 1.570796, 1.512232],accel_mss,speed_ms,0,blend_radius_m)
    |   movel([-0.054523, -1.325129, -2.604023, -0.783238, 1.570796, 1.516273],accel_mss,speed_ms,0,blend_radius_m)
    |   movel([-0.051129, -1.321798, -2.606115, -0.784476, 1.570796, 1.519667],accel_mss,speed_ms,0,blend_radius_m)
    |   movel([-0.045692, -1.317282, -2.608929, -0.786179, 1.570796, 1.525104],accel_mss,speed_ms,0,blend_radius_m)
    |   movel([-0.040005, -1.313397, -2.611327, -0.787665, 1.570796, 1.530791],accel_mss,speed_ms,0,blend_radius_m)
    |   movel([-0.034153, -1.310170, -2.613304, -0.788914, 1.570796, 1.536643],accel_mss,speed_ms,0,blend_radius_m)
    |   movel([-0.028236, -1.307628, -2.614852, -0.789908, 1.570796, 1.542561],accel_mss,speed_ms,0,blend_radius_m)
    |   movel([-0.022348, -1.305795, -2.615963, -0.790631, 1.570796, 1.548449],accel_mss,speed_ms,0,blend_radius_m)
    |   movel([-0.016580, -1.304686, -2.616634, -0.791070, 1.570796, 1.554216],accel_mss,speed_ms,0,blend_radius_m)
    |   movel([-0.011030, -1.304317, -2.616856, -0.791216, 1.570796, 1.559766],accel_mss,speed_ms,0,blend_radius_m)
    |   movel([-0.005791, -1.304700, -2.616625, -0.791064, 1.570796, 1.565005],accel_mss,speed_ms,0,blend_radius_m)
    |   movel([-0.001418, -1.305694, -2.616024, -0.790670, 1.570796, 1.569378],accel_mss,speed_ms,0,blend_radius_m)
    |   movel([0.002673, -1.307080, -2.615185, -0.790124, 1.570796, 1.573469],accel_mss,speed_ms,0,blend_radius_m)
    |   movel([0.006644, -1.308526, -2.614306, -0.789556, 1.570796, 1.577440],accel_mss,speed_ms,0,blend_radius_m)
    |   movel([0.010668, -1.309702, -2.613590, -0.789097, 1.570796, 1.581464],accel_mss,speed_ms,0,blend_radius_m)
    |   movel([0.014918, -1.310286, -2.613234, -0.788870, 1.570796, 1.585715],accel_mss,speed_ms,0,blend_radius_m)
    |   movel([0.017183, -1.310251, -2.613255, -0.788883, 1.570796, 1.587979],accel_mss,speed_ms,0,blend_radius_m)
    |   movel([0.019570, -1.309949, -2.613439, -0.789001, 1.570796, 1.590366],accel_mss,speed_ms,0,blend_radius_m)
    |   movel([0.022104, -1.309335, -2.613814, -0.789240, 1.570796, 1.592900],accel_mss,speed_ms,0,blend_radius_m)
    |   movel([0.024809, -1.308369, -2.614402, -0.789618, 1.570796, 1.595605],accel_mss,speed_ms,0,blend_radius_m)
    |   movel([0.027712, -1.307006, -2.615230, -0.790153, 1.570796, 1.598508],accel_mss,speed_ms,0,blend_radius_m)
    |   movel([0.030836, -1.305204, -2.616321, -0.790864, 1.570796, 1.601633],accel_mss,speed_ms,0,blend_radius_m)
    |   movel([0.033462, -1.303311, -2.617462, -0.791616, 1.570796, 1.604259],accel_mss,speed_ms,0,blend_radius_m)
    |   movel([0.035502, -1.301346, -2.618642, -0.792401, 1.570796, 1.606298],accel_mss,speed_ms,0,blend_radius_m)
    |   movel([0.036986, -1.299357, -2.619831, -0.793201, 1.570796, 1.607782],accel_mss,speed_ms,0,blend_radius_m)
    |   movel([0.037958, -1.297392, -2.621001, -0.793996, 1.570796, 1.608754],accel_mss,speed_ms,0,blend_radius_m)
    |   movel([0.038450, -1.295502, -2.622121, -0.794766, 1.570796, 1.609246],accel_mss,speed_ms,0,blend_radius_m)
    |   movel([0.038495, -1.293743, -2.623160, -0.795486, 1.570796, 1.609292],accel_mss,speed_ms,0,blend_radius_m)
    |   movel([0.038134, -1.292163, -2.624089, -0.796137, 1.570796, 1.608931],accel_mss,speed_ms,0,blend_radius_m)
    |   movel([0.037403, -1.290817, -2.624879, -0.796693, 1.570796, 1.608199],accel_mss,speed_ms,0,blend_radius_m)
    |   movel([0.036339, -1.289760, -2.625497, -0.797132, 1.570796, 1.607135],accel_mss,speed_ms,0,blend_radius_m)
    |   movel([0.034980, -1.289045, -2.625915, -0.797429, 1.570796, 1.605776],accel_mss,speed_ms,0,blend_radius_m)
    |   movel([0.033366, -1.288725, -2.626101, -0.797563, 1.570796, 1.604163],accel_mss,speed_ms,0,blend_radius_m)
    |   movel([0.031539, -1.288853, -2.626027, -0.797510, 1.570796, 1.602335],accel_mss,speed_ms,0,blend_radius_m)
    |   movel([0.029539, -1.289474, -2.625664, -0.797251, 1.570796, 1.600335],accel_mss,speed_ms,0,blend_radius_m)
    |   movel([0.027413, -1.290642, -2.624982, -0.796766, 1.570796, 1.598209],accel_mss,speed_ms,0,blend_radius_m)
    |   movel([0.025201, -1.292403, -2.623948, -0.796037, 1.570796, 1.595998],accel_mss,speed_ms,0,blend_radius_m)
    |   movel([0.022949, -1.294798, -2.622537, -0.795054, 1.570796, 1.593746],accel_mss,speed_ms,0,blend_radius_m)
    |   movel([0.024835, -1.294234, -2.622870, -0.795285, 1.570796, 1.595631],accel_mss,speed_ms,0,blend_radius_m)
    |   movel([0.026385, -1.294077, -2.622963, -0.795349, 1.570796, 1.597182],accel_mss,speed_ms,0,blend_radius_m)
    |   movel([0.027564, -1.294304, -2.622829, -0.795256, 1.570796, 1.598361],accel_mss,speed_ms,0,blend_radius_m)
    |   movel([0.028342, -1.294888, -2.622484, -0.795017, 1.570796, 1.599138],accel_mss,speed_ms,0,blend_radius_m)
    |   movel([0.028683, -1.295809, -2.621940, -0.794641, 1.570796, 1.599479],accel_mss,speed_ms,0,blend_radius_m)
    |   movel([0.028557, -1.297039, -2.621210, -0.794140, 1.570796, 1.599354],accel_mss,speed_ms,0,blend_radius_m)
    |   movel([0.027935, -1.298550, -2.620312, -0.793527, 1.570796, 1.598731],accel_mss,speed_ms,0,blend_radius_m)
    |   movel([0.026784, -1.300320, -2.619256, -0.792813, 1.570796, 1.597581],accel_mss,speed_ms,0,blend_radius_m)
    |   movel([0.024280, -1.303118, -2.617578, -0.791693, 1.570796, 1.595077],accel_mss,speed_ms,0,blend_radius_m)
    |   movel([0.021602, -1.305191, -2.616329, -0.790870, 1.570796, 1.592398],accel_mss,speed_ms,0,blend_radius_m)
    |   movel([0.018815, -1.306593, -2.615480, -0.790316, 1.570796, 1.589612],accel_mss,speed_ms,0,blend_radius_m)
    |   movel([0.016000, -1.307372, -2.615008, -0.790009, 1.570796, 1.586796],accel_mss,speed_ms,0,blend_radius_m)
    |   movel([0.013225, -1.307572, -2.614887, -0.789931, 1.570796, 1.584021],accel_mss,speed_ms,0,blend_radius_m)
    |   movel([0.010566, -1.307233, -2.615092, -0.790064, 1.570796, 1.581362],accel_mss,speed_ms,0,blend_radius_m)
    |   movel([0.008102, -1.306397, -2.615599, -0.790393, 1.570796, 1.578898],accel_mss,speed_ms,0,blend_radius_m)
    |   movel([0.005906, -1.305103, -2.616381, -0.790904, 1.570796, 1.576702],accel_mss,speed_ms,0,blend_radius_m)
    |   movel([0.004062, -1.303381, -2.617420, -0.791588, 1.570796, 1.574859],accel_mss,speed_ms,0,blend_radius_m)
    |   movel([0.002647, -1.301272, -2.618686, -0.792431, 1.570796, 1.573443],accel_mss,speed_ms,0,blend_radius_m)
    |   movel([0.001748, -1.298803, -2.620161, -0.793425, 1.570796, 1.572545],accel_mss,speed_ms,0,blend_radius_m)
    |   movel([0.001450, -1.296012, -2.621819, -0.794558, 1.570796, 1.572246],accel_mss,speed_ms,0,blend_radius_m)
    |   movel([0.001841, -1.292927, -2.623641, -0.795822, 1.570796, 1.572637],accel_mss,speed_ms,0,blend_radius_m)
    |   movel([0.003010, -1.289582, -2.625601, -0.797206, 1.570796, 1.573806],accel_mss,speed_ms,0,blend_radius_m)
    |   movel([0.005052, -1.286011, -2.627679, -0.798699, 1.570796, 1.575848],accel_mss,speed_ms,0,blend_radius_m)
    |   movel([0.008055, -1.282252, -2.629848, -0.800289, 1.570796, 1.578851],accel_mss,speed_ms,0,blend_radius_m)
    |   movel([0.010545, -1.279696, -2.631313, -0.801380, 1.570796, 1.581341],accel_mss,speed_ms,0,blend_radius_m)
    |   movel([0.013182, -1.277305, -2.632676, -0.802408, 1.570796, 1.583978],accel_mss,speed_ms,0,blend_radius_m)
    |   movel([0.015934, -1.275092, -2.633932, -0.803365, 1.570796, 1.586731],accel_mss,speed_ms,0,blend_radius_m)
    |   movel([0.018783, -1.273077, -2.635069, -0.804243, 1.570796, 1.589579],accel_mss,speed_ms,0,blend_radius_m)
    |   movel([0.021695, -1.271275, -2.636082, -0.805032, 1.570796, 1.592491],accel_mss,speed_ms,0,blend_radius_m)
    |   movel([0.024648, -1.269703, -2.636963, -0.805723, 1.570796, 1.595444],accel_mss,speed_ms,0,blend_radius_m)
    |   movel([0.027613, -1.268378, -2.637703, -0.806308, 1.570796, 1.598410],accel_mss,speed_ms,0,blend_radius_m)
    |   movel([0.030563, -1.267314, -2.638295, -0.806780, 1.570796, 1.601360],accel_mss,speed_ms,0,blend_radius_m)
    |   movel([0.033469, -1.266531, -2.638731, -0.807128, 1.570796, 1.604266],accel_mss,speed_ms,0,blend_radius_m)
    |   movel([0.036305, -1.266038, -2.639004, -0.807347, 1.570796, 1.607101],accel_mss,speed_ms,0,blend_radius_m)
    |   movel([0.039042, -1.265856, -2.639105, -0.807428, 1.570796, 1.609838],accel_mss,speed_ms,0,blend_radius_m)
    |   movel([0.041654, -1.265996, -2.639027, -0.807366, 1.570796, 1.612451],accel_mss,speed_ms,0,blend_radius_m)
    |   movel([0.044111, -1.266472, -2.638763, -0.807154, 1.570796, 1.614907],accel_mss,speed_ms,0,blend_radius_m)
    |   movel([0.046390, -1.267293, -2.638307, -0.806789, 1.570796, 1.617186],accel_mss,speed_ms,0,blend_radius_m)
    |   movel([0.048461, -1.268477, -2.637648, -0.806264, 1.570796, 1.619257],accel_mss,speed_ms,0,blend_radius_m)
    |   movel([0.050299, -1.270031, -2.636779, -0.805578, 1.570796, 1.621095],accel_mss,speed_ms,0,blend_radius_m)
    |   movel([0.051489, -1.272144, -2.635594, -0.804650, 1.570796, 1.622286],accel_mss,speed_ms,0,blend_radius_m)
    |   movel([0.052205, -1.274852, -2.634067, -0.803469, 1.570796, 1.623002],accel_mss,speed_ms,0,blend_radius_m)
    |   movel([0.052659, -1.277284, -2.632688, -0.802416, 1.570796, 1.623456],accel_mss,speed_ms,0,blend_radius_m)
    |   movel([0.053064, -1.278582, -2.631949, -0.801858, 1.570796, 1.623860],accel_mss,speed_ms,0,blend_radius_m)
    |   movel([0.054264, -1.278779, -2.631837, -0.801773, 1.570796, 1.625060],accel_mss,speed_ms,0,blend_radius_m)
    |   movel([0.056461, -1.278666, -2.631901, -0.801821, 1.570796, 1.627257],accel_mss,speed_ms,0,blend_radius_m)
    |   movel([0.058885, -1.278544, -2.631971, -0.801874, 1.570796, 1.629681],accel_mss,speed_ms,0,blend_radius_m)
    |   movel([0.060765, -1.278700, -2.631882, -0.801807, 1.570796, 1.631562],accel_mss,speed_ms,0,blend_radius_m)
    |   movel([0.062834, -1.279532, -2.631407, -0.801450, 1.570796, 1.633631],accel_mss,speed_ms,0,blend_radius_m)
    |   movel([0.064472, -1.280680, -2.630751, -0.800959, 1.570796, 1.635268],accel_mss,speed_ms,0,blend_radius_m)
    |   movel([0.065692, -1.282108, -2.629931, -0.800350, 1.570796, 1.636488],accel_mss,speed_ms,0,blend_radius_m)
    |   movel([0.066513, -1.283776, -2.628971, -0.799642, 1.570796, 1.637309],accel_mss,speed_ms,0,blend_radius_m)
    |   movel([0.066955, -1.285648, -2.627889, -0.798852, 1.570796, 1.637752],accel_mss,speed_ms,0,blend_radius_m)
    |   movel([0.067036, -1.287682, -2.626708, -0.797998, 1.570796, 1.637832],accel_mss,speed_ms,0,blend_radius_m)
    |   movel([0.066776, -1.289843, -2.625448, -0.797097, 1.570796, 1.637572],accel_mss,speed_ms,0,blend_radius_m)
    |   movel([0.066191, -1.292094, -2.624130, -0.796165, 1.570796, 1.636988],accel_mss,speed_ms,0,blend_radius_m)
    |   movel([0.065300, -1.294401, -2.622772, -0.795216, 1.570796, 1.636097],accel_mss,speed_ms,0,blend_radius_m)
    |   movel([0.064122, -1.296725, -2.621397, -0.794267, 1.570796, 1.634918],accel_mss,speed_ms,0,blend_radius_m)
    |   movel([0.062673, -1.299035, -2.620023, -0.793331, 1.570796, 1.633469],accel_mss,speed_ms,0,blend_radius_m)
    |   speed_ms = 0.003
    |   movel([0.062673, -1.292173, -2.616738, -0.803478, 1.570796, 1.633469],accel_mss,speed_ms,0,blend_radius_m)
    |   speed_ms = 0.05
    |   movel([0.062673, -1.265901, -2.603322, -0.843166, 1.570796, 1.633469],accel_mss,speed_ms,0,blend_radius_m)
    |   #M_RunCode9
    |   movel([0.079276, -1.257744, -2.607923, -0.846722, 1.570796, 1.650073],accel_mss,speed_ms,0,blend_radius_m)
    |   #M_RunCode3
    |   movel([0.079276, -1.284127, -2.621447, -0.806816, 1.570796, 1.650073],accel_mss,speed_ms,0,blend_radius_m)
    |   speed_ms = 0.003
    |   movel([0.079276, -1.291022, -2.624759, -0.796608, 1.570796, 1.650073],accel_mss,speed_ms,0,blend_radius_m)
    |   speed_ms = 0.02
    |   movel([0.079182, -1.289313, -2.625758, -0.797318, 1.570796, 1.649979],accel_mss,speed_ms,0,blend_radius_m)
    |   movel([0.079578, -1.285585, -2.627926, -0.798879, 1.570796, 1.650374],accel_mss,speed_ms,0,blend_radius_m)
    |   movel([0.079753, -1.282031, -2.629975, -0.800383, 1.570796, 1.650549],accel_mss,speed_ms,0,blend_radius_m)
    |   movel([0.079381, -1.280546, -2.630827, -0.801016, 1.570796, 1.650178],accel_mss,speed_ms,0,blend_radius_m)
    |   movel([0.078497, -1.279378, -2.631495, -0.801516, 1.570796, 1.649293],accel_mss,speed_ms,0,blend_radius_m)
    |   movel([0.079533, -1.279857, -2.631221, -0.801311, 1.570796, 1.650329],accel_mss,speed_ms,0,blend_radius_m)
    |   movel([0.081004, -1.281148, -2.630482, -0.800759, 1.570796, 1.651801],accel_mss,speed_ms,0,blend_radius_m)
    |   movel([0.081818, -1.282779, -2.629545, -0.800065, 1.570796, 1.652614],accel_mss,speed_ms,0,blend_radius_m)
    |   movel([0.082178, -1.284645, -2.628469, -0.799275, 1.570796, 1.652974],accel_mss,speed_ms,0,blend_radius_m)
    |   movel([0.082289, -1.286641, -2.627313, -0.798435, 1.570796, 1.653085],accel_mss,speed_ms,0,blend_radius_m)
    |   movel([0.082574, -1.290622, -2.624993, -0.796774, 1.570796, 1.653370],accel_mss,speed_ms,0,blend_radius_m)
    |   movel([0.083146, -1.292412, -2.623943, -0.796034, 1.570796, 1.653942],accel_mss,speed_ms,0,blend_radius_m)
    |   movel([0.084268, -1.293936, -2.623046, -0.795407, 1.570796, 1.655064],accel_mss,speed_ms,0,blend_radius_m)
    |   movel([0.086018, -1.295241, -2.622276, -0.794873, 1.570796, 1.656814],accel_mss,speed_ms,0,blend_radius_m)
    |   movel([0.087065, -1.295825, -2.621930, -0.794634, 1.570796, 1.657861],accel_mss,speed_ms,0,blend_radius_m)
    |   movel([0.087819, -1.295990, -2.621832, -0.794567, 1.570796, 1.658615],accel_mss,speed_ms,0,blend_radius_m)
    |   movel([0.089062, -1.295029, -2.622401, -0.794959, 1.570796, 1.659858],accel_mss,speed_ms,0,blend_radius_m)
    |   movel([0.090104, -1.294278, -2.622844, -0.795267, 1.570796, 1.660900],accel_mss,speed_ms,0,blend_radius_m)
    |   movel([0.091245, -1.293667, -2.623204, -0.795517, 1.570796, 1.662041],accel_mss,speed_ms,0,blend_radius_m)
    |   movel([0.093544, -1.292886, -2.623664, -0.795839, 1.570796, 1.664341],accel_mss,speed_ms,0,blend_radius_m)
    |   movel([0.095252, -1.292611, -2.623826, -0.795952, 1.570796, 1.666049],accel_mss,speed_ms,0,blend_radius_m)
    |   movel([0.096505, -1.292746, -2.623747, -0.795896, 1.570796, 1.667301],accel_mss,speed_ms,0,blend_radius_m)
    |   movel([0.097444, -1.293201, -2.623479, -0.795709, 1.570796, 1.668240],accel_mss,speed_ms,0,blend_radius_m)
    |   movel([0.098946, -1.294696, -2.622598, -0.795095, 1.570796, 1.669743],accel_mss,speed_ms,0,blend_radius_m)
    |   movel([0.100895, -1.296364, -2.621610, -0.794414, 1.570796, 1.671692],accel_mss,speed_ms,0,blend_radius_m)
    |   movel([0.104110, -1.298008, -2.620635, -0.793747, 1.570796, 1.674906],accel_mss,speed_ms,0,blend_radius_m)
    |   movel([0.107423, -1.299511, -2.619739, -0.793139, 1.570796, 1.678219],accel_mss,speed_ms,0,blend_radius_m)
    |   movel([0.110560, -1.301203, -2.618727, -0.792458, 1.570796, 1.681356],accel_mss,speed_ms,0,blend_radius_m)
    |   movel([0.113253, -1.303396, -2.617411, -0.791582, 1.570796, 1.684050],accel_mss,speed_ms,0,blend_radius_m)
    |   movel([0.114384, -1.304882, -2.616515, -0.790992, 1.570796, 1.685180],accel_mss,speed_ms,0,blend_radius_m)
    |   movel([0.115256, -1.306555, -2.615503, -0.790331, 1.570796, 1.686053],accel_mss,speed_ms,0,blend_radius_m)
    |   movel([0.116468, -1.310252, -2.613254, -0.788883, 1.570796, 1.687264],accel_mss,speed_ms,0,blend_radius_m)
    |   movel([0.117372, -1.314078, -2.610908, -0.787403, 1.570796, 1.688168],accel_mss,speed_ms,0,blend_radius_m)
    |   movel([0.118449, -1.317628, -2.608714, -0.786047, 1.570796, 1.689246],accel_mss,speed_ms,0,blend_radius_m)
    |   movel([0.121104, -1.322927, -2.605407, -0.784054, 1.570796, 1.691901],accel_mss,speed_ms,0,blend_radius_m)
    |   movel([0.122316, -1.325141, -2.604015, -0.783233, 1.570796, 1.693112],accel_mss,speed_ms,0,blend_radius_m)
    |   movel([0.123257, -1.327360, -2.602613, -0.782416, 1.570796, 1.694054],accel_mss,speed_ms,0,blend_radius_m)
    |   movel([0.123798, -1.329795, -2.601066, -0.781528, 1.570796, 1.694594],accel_mss,speed_ms,0,blend_radius_m)
    |   movel([0.123793, -1.332661, -2.599236, -0.780492, 1.570796, 1.694590],accel_mss,speed_ms,0,blend_radius_m)
    |   movel([0.123109, -1.336167, -2.596982, -0.779240, 1.570796, 1.693905],accel_mss,speed_ms,0,blend_radius_m)
    |   movel([0.121617, -1.340512, -2.594165, -0.777711, 1.570796, 1.692413],accel_mss,speed_ms,0,blend_radius_m)
    |   movel([0.120010, -1.344054, -2.591850, -0.776485, 1.570796, 1.690807],accel_mss,speed_ms,0,blend_radius_m)
    |   movel([0.118181, -1.347275, -2.589730, -0.775384, 1.570796, 1.688977],accel_mss,speed_ms,0,blend_radius_m)
    |   movel([0.116146, -1.350191, -2.587799, -0.774399, 1.570796, 1.686942],accel_mss,speed_ms,0,blend_radius_m)
    |   movel([0.113919, -1.352822, -2.586045, -0.773521, 1.570796, 1.684715],accel_mss,speed_ms,0,blend_radius_m)
    |   movel([0.111524, -1.355182, -2.584465, -0.772742, 1.570796, 1.682320],accel_mss,speed_ms,0,blend_radius_m)
    |   movel([0.108974, -1.357288, -2.583048, -0.772053, 1.570796, 1.679770],accel_mss,speed_ms,0,blend_radius_m)
    |   movel([0.106287, -1.359152, -2.581788, -0.771448, 1.570796, 1.677084],accel_mss,speed_ms,0,blend_radius_m)
    |   movel([0.103479, -1.360792, -2.580676, -0.770920, 1.570796, 1.674275],accel_mss,speed_ms,0,blend_radius_m)
    |   movel([0.100570, -1.362219, -2.579706, -0.770464, 1.570796, 1.671366],accel_mss,speed_ms,0,blend_radius_m)
    |   movel([0.097571, -1.363450, -2.578866, -0.770073, 1.570796, 1.668367],accel_mss,speed_ms,0,blend_radius_m)
    |   movel([0.091375, -1.365371, -2.577552, -0.769466, 1.570796, 1.662171],accel_mss,speed_ms,0,blend_radius_m)
    |   movel([0.085030, -1.366656, -2.576669, -0.769064, 1.570796, 1.655826],accel_mss,speed_ms,0,blend_radius_m)
    |   movel([0.078670, -1.367404, -2.576155, -0.768830, 1.570796, 1.649466],accel_mss,speed_ms,0,blend_radius_m)
    |   movel([0.072831, -1.367616, -2.576008, -0.768764, 1.570796, 1.643627],accel_mss,speed_ms,0,blend_radius_m)
    |   movel([0.065389, -1.367790, -2.575889, -0.768710, 1.570796, 1.636186],accel_mss,speed_ms,0,blend_radius_m)
    |   movel([0.057017, -1.368376, -2.575485, -0.768528, 1.570796, 1.627813],accel_mss,speed_ms,0,blend_radius_m)
    |   movel([0.052698, -1.368956, -2.575085, -0.768348, 1.570796, 1.623495],accel_mss,speed_ms,0,blend_radius_m)
    |   movel([0.048406, -1.369796, -2.574504, -0.768089, 1.570796, 1.619202],accel_mss,speed_ms,0,blend_radius_m)
    |   movel([0.044238, -1.370942, -2.573710, -0.767737, 1.570796, 1.615034],accel_mss,speed_ms,0,blend_radius_m)
    |   movel([0.040279, -1.372440, -2.572669, -0.767279, 1.570796, 1.611075],accel_mss,speed_ms,0,blend_radius_m)
    |   movel([0.036623, -1.374335, -2.571349, -0.766705, 1.570796, 1.607420],accel_mss,speed_ms,0,blend_radius_m)
    |   movel([0.033366, -1.376665, -2.569718, -0.766006, 1.570796, 1.604162],accel_mss,speed_ms,0,blend_radius_m)
    |   movel([0.031912, -1.378007, -2.568775, -0.765607, 1.570796, 1.602708],accel_mss,speed_ms,0,blend_radius_m)
    |   movel([0.030592, -1.379474, -2.567741, -0.765174, 1.570796, 1.601389],accel_mss,speed_ms,0,blend_radius_m)
    |   movel([0.029416, -1.381068, -2.566615, -0.764706, 1.570796, 1.600212],accel_mss,speed_ms,0,blend_radius_m)
    |   movel([0.028394, -1.382796, -2.565389, -0.764204, 1.570796, 1.599190],accel_mss,speed_ms,0,blend_radius_m)
    |   movel([0.027538, -1.384663, -2.564061, -0.763666, 1.570796, 1.598334],accel_mss,speed_ms,0,blend_radius_m)
    |   movel([0.026856, -1.386673, -2.562624, -0.763092, 1.570796, 1.597652],accel_mss,speed_ms,0,blend_radius_m)
